C05459=1123.392,111.810,-57.603,-179.804,8.191,149.512
C05460=1123.397,111.561,-57.584,-179.806,8.187,149.511
C05461=1123.401,111.312,-57.565,-179.808,8.184,149.511
C05462=1123.406,111.062,-57.545,-179.809,8.181,149.511
C05463=1123.411,110.813,-57.526,-179.812,8.177,149.510
C05464=1123.416,110.564,-57.506,-179.814,8.173,149.510
C05465=1123.421,110.314,-57.487,-179.817,8.169,149.510
C05466=1123.426,110.066,-57.468,-179.819,8.165,149.510
C05467=1123.430,109.816,-57.448,-179.822,8.161,149.510
C05468=1123.436,109.567,-57.429,-179.824,8.158,149.509
C05469=1123.440,109.318,-57.409,-179.826,8.154,149.509
C05470=1123.444,109.068,-57.390,-179.828,8.150,149.509
C05471=1123.450,108.820,-57.371,-179.830,8.146,149.509
C05472=1123.455,108.570,-57.351,-179.833,8.142,149.508
C05473=1123.460,108.321,-57.332,-179.835,8.138,149.508
C05474=1123.464,108.072,-57.313,-179.838,8.134,149.508
C05475=1123.469,107.823,-57.294,-179.840,8.131,149.508
C05476=1123.474,107.573,-57.274,-179.843,8.126,149.508
C05477=1123.478,107.324,-57.255,-179.845,8.123,149.507
C05478=1123.483,107.075,-57.236,-179.846,8.119,149.507
C05479=1123.488,106.826,-57.216,-179.849,8.115,149.507
C05480=1123.493,106.577,-57.198,-179.851,8.111,149.506
C05481=1123.498,106.327,-57.178,-179.854,8.107,149.506
C05482=1123.503,106.078,-57.159,-179.856,8.103,149.506
C05483=1123.507,105.829,-57.140,-179.857,8.100,149.506
C05484=1123.512,105.580,-57.121,-179.860,8.095,149.505
C05485=1123.516,105.331,-57.102,-179.862,8.092,149.505
C05486=1123.522,105.081,-57.083,-179.864,8.088,149.505
C05487=1123.527,104.832,-57.064,-179.866,8.084,149.505
C05488=1123.531,104.583,-57.045,-179.868,8.080,149.504
C05489=1123.536,104.334,-57.025,-179.870,8.076,149.504
C05490=1123.541,104.084,-57.007,-179.873,8.072,149.504
C05491=1123.546,103.870,-56.991,-179.874,8.069,149.503
C05492=1123.549,103.655,-56.974,-179.876,8.066,149.503
C05493=1123.553,103.441,-56.957,-179.878,8.062,149.503
C05494=1123.557,103.227,-56.941,-179.880,8.058,149.503
C05495=1123.562,103.012,-56.925,-179.881,8.056,149.502
C05496=1123.566,102.798,-56.909,-179.883,8.052,149.502
C05497=1123.570,102.582,-56.892,-179.885,8.048,149.502
C05498=1123.574,102.368,-56.876,-179.886,8.046,149.501
C05499=1123.579,102.119,-56.857,-179.889,8.041,149.501
C05500=1123.583,101.870,-56.838,-179.891,8.037,149.501
C05501=1123.589,101.620,-56.820,-179.892,8.033,149.500
C05502=1123.594,101.372,-56.801,-179.894,8.030,149.500
C05503=1123.598,101.122,-56.781,-179.897,8.025,149.500
C05504=1123.603,100.873,-56.763,-179.899,8.022,149.500
C05505=1123.608,100.623,-56.744,-179.900,8.018,149.499
C05506=1123.613,100.374,-56.726,-179.902,8.014,149.499
C05507=1123.618,100.125,-56.707,-179.905,8.010,149.498
C05508=1123.623,99.875,-56.688,-179.906,8.006,149.498
C05509=1123.627,99.627,-56.669,-179.908,8.002,149.498
C05510=1123.632,99.377,-56.651,-179.910,7.998,149.497
C05511=1123.637,99.128,-56.632,-179.911,7.995,149.497
C05512=1123.642,98.878,-56.613,-179.914,7.990,149.497
C05513=1123.646,98.629,-56.594,-179.916,7.986,149.496
C05514=1123.651,98.380,-56.576,-179.917,7.982,149.496
C05515=1123.657,98.131,-56.557,-179.919,7.979,149.495
C05516=1123.661,97.881,-56.539,-179.921,7.975,149.495
C05517=1123.666,97.632,-56.521,-179.923,7.971,149.495
C05518=1123.671,97.383,-56.501,-179.925,7.967,149.494
C05519=1123.676,97.133,-56.483,-179.926,7.963,149.494
C05520=1123.680,96.885,-56.464,-179.928,7.959,149.494
C05521=1123.686,96.635,-56.446,-179.930,7.955,149.493
C05522=1123.690,96.385,-56.427,-179.932,7.951,149.493
C05523=1123.695,96.137,-56.409,-179.933,7.947,149.492
C05524=1123.700,95.888,-56.391,-179.935,7.944,149.492
C05525=1123.705,95.638,-56.372,-179.936,7.940,149.492
C05526=1123.709,95.389,-56.353,-179.938,7.936,149.491
C05527=1123.714,95.140,-56.335,-179.940,7.932,149.491
C05528=1123.720,94.890,-56.317,-179.942,7.927,149.490
C05529=1123.724,94.640,-56.298,-179.943,7.923,149.490
C05530=1123.729,94.392,-56.279,-179.945,7.919,149.489
C05531=1123.734,94.143,-56.261,-179.947,7.916,149.489
C05532=1123.739,93.894,-56.244,-179.948,7.912,149.489
C05533=1123.744,93.643,-56.225,-179.950,7.908,149.488
C05534=1123.748,93.395,-56.206,-179.951,7.904,149.488
C05535=1123.753,93.146,-56.188,-179.953,7.900,149.487
C05536=1123.758,92.896,-56.170,-179.955,7.896,149.487
C05537=1123.762,92.647,-56.152,-179.956,7.892,149.486
C05538=1123.768,92.397,-56.133,-179.958,7.888,149.486
C05539=1123.773,92.148,-56.115,-179.959,7.884,149.486
C05540=1123.778,91.899,-56.096,-179.961,7.881,149.485
C05541=1123.783,91.650,-56.078,-179.963,7.877,149.485
C05542=1123.787,91.400,-56.060,-179.964,7.873,149.484
C05543=1123.792,91.151,-56.042,-179.966,7.869,149.484
C05544=1123.797,90.902,-56.023,-179.967,7.865,149.483
C05545=1123.802,90.652,-56.005,-179.968,7.862,149.483
C05546=1123.807,90.403,-55.987,-179.970,7.858,149.482
C05547=1123.811,90.189,-55.972,-179.972,7.854,149.482
C05548=1123.815,89.974,-55.956,-179.973,7.851,149.482
C05549=1123.819,89.760,-55.941,-179.974,7.848,149.481
C05550=1123.823,89.545,-55.925,-179.975,7.844,149.481
C05551=1123.828,89.330,-55.909,-179.976,7.841,149.480
C05552=1123.832,89.115,-55.894,-179.978,7.837,149.480
C05553=1123.837,88.901,-55.878,-179.979,7.834,149.480
C05554=1123.840,88.686,-55.862,-179.980,7.831,149.479
C05555=1123.845,88.437,-55.844,-179.981,7.827,149.479
C05556=1123.850,88.187,-55.826,-179.983,7.823,149.478
C05557=1123.854,87.938,-55.808,-179.984,7.819,149.478
C05558=1123.860,87.688,-55.791,-179.986,7.815,149.477
C05559=1123.865,87.439,-55.773,-179.987,7.812,149.477
C05560=1123.870,87.190,-55.755,-179.988,7.808,149.476
C05561=1123.874,86.941,-55.737,-179.990,7.804,149.476
C05562=1123.879,86.692,-55.719,-179.991,7.800,149.475
C05563=1123.884,86.443,-55.701,-179.992,7.796,149.475
C05564=1123.889,86.193,-55.683,-179.993,7.793,149.474
C05565=1123.893,85.943,-55.665,-179.995,7.788,149.474
C05566=1123.898,85.694,-55.647,-179.996,7.784,149.473
C05567=1123.903,85.445,-55.629,-179.998,7.781,149.473
C05568=1123.909,85.195,-55.611,-179.998,7.777,149.472
C05569=1123.913,84.946,-55.593,-180.000,7.773,149.472
C05570=1123.918,84.697,-55.575,179.999,7.769,149.471
C05571=1123.923,84.448,-55.557,179.997,7.765,149.471
C05572=1123.928,84.199,-55.539,179.996,7.762,149.470
C05573=1123.933,83.949,-55.521,179.995,7.758,149.470
C05574=1123.938,83.700,-55.504,179.994,7.754,149.469
C05575=1123.943,83.450,-55.486,179.993,7.751,149.469
C05576=1123.948,83.201,-55.468,179.992,7.746,149.468
C05577=1123.952,82.952,-55.451,179.990,7.742,149.468
C05578=1123.958,82.703,-55.434,179.990,7.739,149.467
C05579=1123.962,82.453,-55.416,179.988,7.735,149.467
C05580=1123.967,82.204,-55.398,179.986,7.731,149.466
C05581=1123.972,81.955,-55.380,179.986,7.728,149.466
C05582=1123.977,81.705,-55.362,179.984,7.724,149.465
C05583=1123.982,81.455,-55.344,179.984,7.720,149.465
C05584=1123.986,81.207,-55.327,179.982,7.716,149.464
C05585=1123.991,80.957,-55.309,179.981,7.712,149.463
C05586=1123.996,80.708,-55.291,179.980,7.709,149.463
C05587=1124.001,80.458,-55.273,179.979,7.705,149.462
C05588=1124.006,80.209,-55.256,179.978,7.702,149.462
C05589=1124.011,79.959,-55.238,179.977,7.697,149.461
C05590=1124.016,79.711,-55.221,179.976,7.694,149.461
C05591=1124.021,79.462,-55.204,179.975,7.690,149.460
C05592=1124.026,79.212,-55.186,179.974,7.687,149.460
C05593=1124.031,78.963,-55.168,179.973,7.682,149.459
C05594=1124.036,78.713,-55.151,179.972,7.679,149.459
C05595=1124.040,78.464,-55.133,179.971,7.675,149.458
C05596=1124.046,78.215,-55.116,179.970,7.672,149.457
C05597=1124.050,77.966,-55.098,179.969,7.668,149.457
C05598=1124.056,77.716,-55.081,179.968,7.664,149.456
C05599=1124.061,77.467,-55.063,179.966,7.660,149.456
C05600=1124.065,77.218,-55.045,179.966,7.657,149.455
C05601=1124.070,76.968,-55.028,179.964,7.653,149.455
C05602=1124.075,76.719,-55.010,179.964,7.649,149.454
C05603=1124.079,76.503,-54.996,179.963,7.646,149.454
C05604=1124.083,76.289,-54.981,179.961,7.642,149.453
C05605=1124.087,76.075,-54.966,179.960,7.639,149.453
C05606=1124.092,75.860,-54.951,179.959,7.635,149.453
C05607=1124.096,75.645,-54.936,179.958,7.632,149.452
C05608=1124.100,75.430,-54.920,179.957,7.629,149.452
C05609=1124.105,75.215,-54.906,179.955,7.625,149.451
C05610=1124.109,75.001,-54.891,179.954,7.622,149.451
C05611=1124.114,74.751,-54.874,179.953,7.618,149.450
C05612=1124.119,74.502,-54.856,179.951,7.614,149.450
C05613=1124.123,74.253,-54.839,179.950,7.610,149.450
C05614=1124.128,74.003,-54.821,179.948,7.606,149.449
C05615=1124.133,73.754,-54.804,179.947,7.602,149.448
C05616=1124.138,73.504,-54.787,179.945,7.598,149.448
C05617=1124.143,73.255,-54.769,179.944,7.594,149.448
C05618=1124.149,73.006,-54.752,179.942,7.590,149.447
C05619=1124.153,72.756,-54.736,179.941,7.586,149.447
C05620=1124.158,72.507,-54.718,179.939,7.582,149.446
C05621=1124.162,72.258,-54.701,179.938,7.578,149.446
C05622=1124.168,72.008,-54.684,179.937,7.574,149.445
C05623=1124.173,71.759,-54.666,179.935,7.570,149.445
C05624=1124.177,71.509,-54.649,179.934,7.566,149.444
C05625=1124.183,71.260,-54.632,179.932,7.562,149.444
C05626=1124.187,71.011,-54.615,179.931,7.558,149.443
C05627=1124.192,70.762,-54.598,179.929,7.554,149.443
C05628=1124.197,70.512,-54.581,179.928,7.550,149.442
C05629=1124.202,70.262,-54.564,179.926,7.546,149.442
C05630=1124.207,70.014,-54.546,179.926,7.543,149.441
C05631=1124.212,69.764,-54.529,179.924,7.539,149.441
C05632=1124.217,69.514,-54.512,179.923,7.535,149.440
C05633=1124.222,69.265,-54.496,179.921,7.531,149.440
C05634=1124.227,69.015,-54.478,179.920,7.527,149.439
C05635=1124.232,68.767,-54.461,179.918,7.523,149.439
C05636=1124.237,68.517,-54.444,179.917,7.519,149.438
C05637=1124.241,68.268,-54.427,179.916,7.515,149.438
C05638=1124.247,68.018,-54.410,179.914,7.511,149.437
C05639=1124.252,67.769,-54.394,179.912,7.507,149.437
C05640=1124.256,67.520,-54.377,179.911,7.503,149.436
C05641=1124.261,67.270,-54.360,179.910,7.499,149.436
C05642=1124.265,67.021,-54.342,179.908,7.495,149.435
C05643=1124.271,66.772,-54.326,179.907,7.491,149.435
C05644=1124.276,66.522,-54.309,179.906,7.487,149.434
C05645=1124.281,66.273,-54.292,179.904,7.483,149.434
C05646=1124.285,66.023,-54.275,179.903,7.478,149.433
C05647=1124.291,65.774,-54.259,179.901,7.475,149.433
C05648=1124.296,65.525,-54.241,179.900,7.471,149.432
C05649=1124.300,65.275,-54.225,179.899,7.466,149.432
C05650=1124.306,65.026,-54.208,179.898,7.463,149.431
C05651=1124.311,64.777,-54.191,179.896,7.459,149.431
C05652=1124.315,64.527,-54.174,179.895,7.455,149.430
C05653=1124.321,64.278,-54.158,179.893,7.451,149.430
C05654=1124.325,64.028,-54.141,179.892,7.447,149.429
C05655=1124.330,63.779,-54.124,179.891,7.443,149.429
C05656=1124.335,63.529,-54.107,179.889,7.439,149.428
C05657=1124.340,63.280,-54.091,179.888,7.435,149.428
C05658=1124.345,63.031,-54.074,179.887,7.431,149.427
C05659=1124.350,62.816,-54.060,179.886,7.428,149.427
C05660=1124.353,62.601,-54.046,179.884,7.424,149.426
C05661=1124.358,62.386,-54.031,179.883,7.421,149.426
C05662=1124.362,62.172,-54.017,179.882,7.417,149.426
C05663=1124.366,61.956,-54.003,179.881,7.414,149.425
C05664=1124.370,61.741,-53.988,179.880,7.411,149.425
C05665=1124.375,61.527,-53.973,179.878,7.407,149.424
C05666=1124.379,61.312,-53.959,179.877,7.403,149.424
C05667=1124.385,61.062,-53.943,179.876,7.400,149.423
C05668=1124.389,60.813,-53.927,179.874,7.395,149.423
C05669=1124.394,60.563,-53.910,179.873,7.391,149.422
C05670=1124.399,60.315,-53.894,179.871,7.387,149.422
C05671=1124.404,60.065,-53.876,179.870,7.383,149.421
C05672=1124.409,59.816,-53.860,179.869,7.379,149.421
C05673=1124.414,59.566,-53.844,179.868,7.375,149.420
C05674=1124.418,59.317,-53.827,179.866,7.371,149.420
C05675=1124.423,59.068,-53.811,179.864,7.367,149.419
C05676=1124.429,58.818,-53.794,179.863,7.363,149.419
C05677=1124.434,58.569,-53.778,179.862,7.359,149.418
C05678=1124.438,58.319,-53.762,179.861,7.355,149.418
C05679=1124.444,58.070,-53.745,179.859,7.351,149.417
C05680=1124.448,57.820,-53.729,179.858,7.348,149.417
C05681=1124.453,57.571,-53.713,179.857,7.343,149.416
C05682=1124.459,57.322,-53.696,179.856,7.339,149.416
C05683=1124.463,57.071,-53.680,179.854,7.335,149.415
C05684=1124.469,56.823,-53.663,179.853,7.331,149.415
C05685=1124.473,56.573,-53.647,179.852,7.327,149.414
C05686=1124.478,56.324,-53.631,179.850,7.323,149.414
C05687=1124.483,56.074,-53.615,179.849,7.319,149.413
C05688=1124.488,55.826,-53.598,179.848,7.315,149.412
C05689=1124.493,55.575,-53.582,179.846,7.311,149.412
C05690=1124.499,55.326,-53.565,179.845,7.307,149.411
C05691=1124.503,55.076,-53.549,179.843,7.303,149.411
C05692=1124.508,54.827,-53.533,179.842,7.298,149.410
C05693=1124.513,54.577,-53.517,179.841,7.294,149.410
C05694=1124.518,54.329,-53.501,179.840,7.290,149.409
C05695=1124.523,54.079,-53.484,179.838,7.286,149.409
C05696=1124.528,53.830,-53.469,179.837,7.282,149.408
C05697=1124.533,53.580,-53.452,179.835,7.278,149.408
C05698=1124.538,53.331,-53.436,179.834,7.274,149.407
C05699=1124.542,53.081,-53.420,179.833,7.271,149.407
C05700=1124.548,52.832,-53.404,179.832,7.266,149.406
C05701=1124.552,52.582,-53.387,179.831,7.262,149.406
C05702=1124.558,52.333,-53.372,179.830,7.258,149.405
C05703=1124.563,52.084,-53.356,179.828,7.254,149.405
C05704=1124.568,51.834,-53.340,179.827,7.250,149.404
C05705=1124.573,51.585,-53.324,179.825,7.246,149.403
C05706=1124.577,51.335,-53.307,179.824,7.242,149.403
C05707=1124.583,51.086,-53.292,179.823,7.238,149.402
C05708=1124.587,50.836,-53.275,179.822,7.233,149.402
C05709=1124.593,50.587,-53.259,179.820,7.230,149.401
C05710=1124.598,50.338,-53.244,179.819,7.225,149.401
C05711=1124.603,50.088,-53.227,179.817,7.221,149.400
C05712=1124.608,49.839,-53.212,179.816,7.217,149.400
C05713=1124.613,49.589,-53.196,179.815,7.213,149.399
C05714=1124.618,49.340,-53.179,179.814,7.209,149.398
C05715=1124.622,49.125,-53.166,179.813,7.206,149.398
C05716=1124.626,48.910,-53.152,179.811,7.202,149.398
C05717=1124.630,48.695,-53.139,179.811,7.198,149.397
C05718=1124.634,48.480,-53.125,179.810,7.195,149.397
C05719=1124.639,48.265,-53.111,179.808,7.191,149.396
C05720=1124.643,48.050,-53.098,179.807,7.188,149.396
C05721=1124.648,47.835,-53.084,179.806,7.184,149.395
C05722=1124.652,47.620,-53.071,179.805,7.181,149.395
C05723=1124.657,47.371,-53.054,179.804,7.177,149.394
C05724=1124.662,47.121,-53.039,179.803,7.172,149.394
C05725=1124.667,46.872,-53.024,179.802,7.168,149.393
C05726=1124.672,46.622,-53.008,179.800,7.164,149.392
C05727=1124.677,46.373,-52.991,179.799,7.160,149.392
C05728=1124.682,46.124,-52.976,179.798,7.156,149.391
C05729=1124.687,45.874,-52.960,179.796,7.152,149.391
C05730=1124.692,45.624,-52.944,179.795,7.147,149.390
C05731=1124.697,45.375,-52.929,179.794,7.143,149.390
C05732=1124.702,45.125,-52.913,179.793,7.139,149.389
C05733=1124.707,44.876,-52.897,179.792,7.135,149.388
C05734=1124.712,44.627,-52.881,179.790,7.131,149.388
C05735=1124.716,44.377,-52.866,179.789,7.127,149.387
C05736=1124.722,44.128,-52.850,179.788,7.122,149.387
C05737=1124.727,43.878,-52.835,179.786,7.118,149.386
C05738=1124.732,43.629,-52.819,179.785,7.114,149.386
C05739=1124.736,43.379,-52.804,179.784,7.110,149.385
C05740=1124.742,43.130,-52.788,179.783,7.106,149.385
C05741=1124.747,42.880,-52.773,179.782,7.102,149.384
C05742=1124.753,42.631,-52.757,179.781,7.098,149.383
C05743=1124.757,42.381,-52.742,179.780,7.094,149.383
C05744=1124.762,42.132,-52.726,179.779,7.090,149.382
C05745=1124.767,41.882,-52.711,179.777,7.085,149.382
C05746=1124.772,41.633,-52.696,179.776,7.082,149.381
C05747=1124.777,41.383,-52.680,179.775,7.077,149.380
C05748=1124.782,41.134,-52.664,179.774,7.073,149.380
C05749=1124.787,40.885,-52.649,179.773,7.069,149.379
C05750=1124.792,40.635,-52.634,179.771,7.065,149.379
C05751=1124.797,40.385,-52.618,179.770,7.060,149.378
C05752=1124.802,40.136,-52.603,179.769,7.056,149.377
C05753=1124.807,39.887,-52.587,179.768,7.052,149.377
C05754=1124.813,39.637,-52.571,179.766,7.048,149.376
C05755=1124.817,39.388,-52.556,179.765,7.044,149.376
C05756=1124.823,39.139,-52.541,179.764,7.039,149.375
C05757=1124.827,38.889,-52.525,179.763,7.035,149.374
C05758=1124.832,38.640,-52.510,179.762,7.031,149.374
C05759=1124.837,38.390,-52.494,179.761,7.027,149.373
C05760=1124.842,38.141,-52.480,179.759,7.022,149.373
C05761=1124.848,37.891,-52.464,179.758,7.018,149.372
C05762=1124.852,37.642,-52.449,179.757,7.014,149.371
C05763=1124.857,37.392,-52.433,179.756,7.010,149.371
C05764=1124.863,37.143,-52.418,179.755,7.006,149.370
C05765=1124.868,36.893,-52.404,179.754,7.001,149.370
C05766=1124.873,36.643,-52.388,179.753,6.997,149.369
C05767=1124.878,36.394,-52.373,179.752,6.993,149.368
C05768=1124.883,36.145,-52.357,179.750,6.988,149.368
C05769=1124.888,35.896,-52.342,179.749,6.984,149.367
C05770=1124.893,35.645,-52.327,179.748,6.980,149.367
C05771=1124.897,35.430,-52.314,179.747,6.976,149.366
C05772=1124.902,35.215,-52.301,179.746,6.973,149.366
C05773=1124.905,35.001,-52.288,179.745,6.969,149.365
C05774=1124.910,34.786,-52.275,179.744,6.965,149.364
C05775=1124.914,34.571,-52.262,179.743,6.962,149.364
C05776=1124.919,34.356,-52.249,179.742,6.958,149.363
C05777=1124.923,34.141,-52.236,179.741,6.954,149.363
C05778=1124.928,33.926,-52.223,179.740,6.950,149.362
C05779=1124.933,33.676,-52.209,179.739,6.946,149.362
C05780=1124.938,33.427,-52.193,179.738,6.942,149.361
C05781=1124.943,33.178,-52.178,179.737,6.937,149.360
C05782=1124.947,32.927,-52.163,179.736,6.933,149.360
C05783=1124.953,32.678,-52.148,179.735,6.929,149.359
C05784=1124.957,32.429,-52.133,179.733,6.925,149.359
C05785=1124.963,32.179,-52.118,179.732,6.920,149.358
C05786=1124.968,31.930,-52.103,179.731,6.916,149.357
C05787=1124.973,31.680,-52.089,179.730,6.912,149.357
C05788=1124.978,31.430,-52.073,179.729,6.908,149.356
C05789=1124.983,31.181,-52.059,179.728,6.903,149.355
C05790=1124.988,30.931,-52.043,179.727,6.899,149.355
C05791=1124.993,30.682,-52.028,179.726,6.895,149.354
C05792=1124.998,30.433,-52.014,179.725,6.890,149.353
C05793=1125.003,30.183,-51.998,179.724,6.886,149.353
C05794=1125.008,29.933,-51.984,179.722,6.882,149.352
C05795=1125.013,29.684,-51.969,179.721,6.877,149.352
C05796=1125.019,29.434,-51.954,179.720,6.873,149.351
C05797=1125.023,29.185,-51.939,179.719,6.869,149.350
C05798=1125.028,28.935,-51.925,179.718,6.864,149.350
C05799=1125.034,28.686,-51.909,179.717,6.860,149.349
C05800=1125.038,28.436,-51.895,179.716,6.856,149.348
C05801=1125.043,28.187,-51.881,179.715,6.851,149.348
C05802=1125.048,27.938,-51.866,179.714,6.847,149.347
C05803=1125.054,27.688,-51.851,179.713,6.843,149.346
C05804=1125.058,27.438,-51.836,179.712,6.839,149.346
C05805=1125.063,27.189,-51.822,179.711,6.834,149.345
C05806=1125.069,26.939,-51.807,179.710,6.829,149.344
C05807=1125.074,26.690,-51.792,179.709,6.824,149.344
C05808=1125.079,26.440,-51.777,179.708,6.820,149.343
C05809=1125.084,26.191,-51.764,179.707,6.816,149.342
C05810=1125.089,25.942,-51.749,179.705,6.811,149.342
C05811=1125.095,25.692,-51.734,179.704,6.807,149.341
C05812=1125.100,25.442,-51.719,179.703,6.803,149.340
C05813=1125.104,25.193,-51.704,179.702,6.798,149.340
C05814=1125.109,24.943,-51.690,179.701,6.794,149.339
C05815=1125.115,24.693,-51.675,179.701,6.789,149.338
C05816=1125.119,24.444,-51.660,179.700,6.785,149.337
C05817=1125.124,24.194,-51.646,179.699,6.781,149.337
C05818=1125.129,23.945,-51.632,179.698,6.777,149.336
C05819=1125.134,23.695,-51.617,179.696,6.772,149.335
C05820=1125.140,23.447,-51.603,179.695,6.768,149.335
C05821=1125.145,23.197,-51.588,179.695,6.763,149.334
C05822=1125.150,22.947,-51.574,179.694,6.759,149.333
C05823=1125.155,22.697,-51.559,179.692,6.754,149.333
C05824=1125.160,22.447,-51.545,179.691,6.749,149.332
C05825=1125.165,22.198,-51.530,179.690,6.745,149.331
C05826=1125.170,21.949,-51.516,179.689,6.740,149.331
C05827=1125.175,21.733,-51.504,179.689,6.737,149.330
C05828=1125.179,21.518,-51.491,179.688,6.733,149.329
C05829=1125.183,21.303,-51.479,179.687,6.729,149.329
C05830=1125.187,21.088,-51.466,179.686,6.725,149.328
C05831=1125.192,20.873,-51.454,179.686,6.722,149.327
C05832=1125.196,20.658,-51.442,179.684,6.718,149.327
C05833=1125.201,20.442,-51.429,179.684,6.714,149.326
C05834=1125.205,20.228,-51.417,179.683,6.710,149.326
C05835=1125.210,19.978,-51.403,179.682,6.705,149.325
C05836=1125.215,19.729,-51.389,179.681,6.701,149.324
C05837=1125.220,19.479,-51.375,179.680,6.696,149.324
C05838=1125.225,19.230,-51.360,179.679,6.692,149.323
C05839=1125.230,18.980,-51.346,179.678,6.688,149.322
C05840=1125.235,18.730,-51.332,179.677,6.683,149.321
C05841=1125.241,18.481,-51.318,179.676,6.678,149.321
C05842=1125.246,18.232,-51.304,179.675,6.674,149.320
C05843=1125.251,17.982,-51.289,179.674,6.669,149.319
C05844=1125.256,17.732,-51.275,179.673,6.665,149.319
C05845=1125.261,17.483,-51.261,179.672,6.660,149.318
C05846=1125.266,17.233,-51.247,179.671,6.656,149.317
C05847=1125.271,16.984,-51.233,179.670,6.651,149.316
C05848=1125.276,16.734,-51.218,179.670,6.647,149.315
C05849=1125.282,16.485,-51.204,179.669,6.642,149.315
C05850=1125.287,16.235,-51.190,179.667,6.637,149.314
C05851=1125.291,15.986,-51.176,179.667,6.632,149.313
C05852=1125.296,15.736,-51.162,179.666,6.628,149.313
C05853=1125.302,15.487,-51.148,179.665,6.623,149.312
C05854=1125.307,15.237,-51.133,179.664,6.619,149.311
C05855=1125.312,14.987,-51.119,179.663,6.615,149.310
C05856=1125.317,14.738,-51.105,179.662,6.610,149.310
C05857=1125.323,14.488,-51.092,179.661,6.606,149.309
C05858=1125.327,14.239,-51.078,179.660,6.600,149.308
C05859=1125.332,13.989,-51.064,179.659,6.596,149.307
C05860=1125.337,13.740,-51.050,179.659,6.591,149.307
C05861=1125.342,13.490,-51.035,179.658,6.587,149.306
C05862=1125.347,13.241,-51.021,179.657,6.582,149.305
C05863=1125.353,12.991,-51.008,179.656,6.578,149.304
C05864=1125.358,12.741,-50.994,179.655,6.573,149.304
C05865=1125.362,12.492,-50.980,179.654,6.568,149.303
C05866=1125.368,12.243,-50.966,179.653,6.563,149.302
C05867=1125.373,11.992,-50.953,179.652,6.559,149.301
C05868=1125.378,11.743,-50.938,179.652,6.554,149.300
C05869=1125.384,11.494,-50.924,179.651,6.549,149.300
C05870=1125.389,11.244,-50.910,179.650,6.545,149.299
C05871=1125.393,10.994,-50.897,179.649,6.540,149.298
C05872=1125.399,10.745,-50.883,179.648,6.535,149.297
C05873=1125.404,10.495,-50.869,179.647,6.531,149.297
C05874=1125.410,10.246,-50.856,179.646,6.526,149.296
C05875=1125.414,9.996,-50.842,179.646,6.522,149.295
C05876=1125.419,9.747,-50.828,179.645,6.517,149.294
C05877=1125.425,9.497,-50.815,179.644,6.512,149.293
C05878=1125.430,9.247,-50.800,179.643,6.507,149.293
C05879=1125.434,8.999,-50.787,179.642,6.502,149.292
C05880=1125.440,8.748,-50.773,179.641,6.498,149.291
C05881=1125.445,8.498,-50.759,179.641,6.493,149.290
C05882=1125.450,8.249,-50.746,179.640,6.488,149.289
C05883=1125.455,8.034,-50.734,179.639,6.484,149.289
C05884=1125.459,7.818,-50.723,179.639,6.481,149.288
C05885=1125.463,7.603,-50.711,179.639,6.477,149.287
C05886=1125.467,7.388,-50.699,179.638,6.472,149.286
C05887=1125.473,7.173,-50.687,179.638,6.468,149.286
C05888=1125.477,6.958,-50.676,179.638,6.465,149.285
C05889=1125.481,6.742,-50.664,179.637,6.461,149.284
C05890=1125.485,6.527,-50.652,179.637,6.457,149.283
C05891=1125.491,6.278,-50.638,179.637,6.453,149.282
C05892=1125.495,6.028,-50.625,179.636,6.448,149.282
C05893=1125.500,5.778,-50.611,179.635,6.444,149.281
C05894=1125.506,5.529,-50.598,179.635,6.439,149.280
C05895=1125.510,5.279,-50.584,179.635,6.435,149.279
C05896=1125.516,5.030,-50.571,179.634,6.430,149.278
C05897=1125.521,4.780,-50.557,179.634,6.426,149.277
C05898=1125.526,4.531,-50.544,179.633,6.421,149.277
C05899=1125.531,4.281,-50.530,179.633,6.416,149.276
C05900=1125.536,4.032,-50.517,179.632,6.413,149.275
C05901=1125.541,3.782,-50.503,179.632,6.408,149.274
C05902=1125.547,3.532,-50.490,179.631,6.403,149.273
C05903=1125.551,3.283,-50.476,179.631,6.398,149.272
C05904=1125.557,3.033,-50.463,179.630,6.394,149.271
C05905=1125.562,2.783,-50.450,179.630,6.390,149.271
C05906=1125.567,2.534,-50.436,179.629,6.385,149.270
C05907=1125.572,2.284,-50.423,179.629,6.381,149.269
C05908=1125.577,2.035,-50.409,179.628,6.376,149.268
C05909=1125.583,1.785,-50.396,179.627,6.371,149.267
C05910=1125.588,1.536,-50.383,179.628,6.367,149.266
C05911=1125.593,1.287,-50.369,179.627,6.363,149.266
C05912=1125.598,1.037,-50.356,179.626,6.358,149.265
C05913=1125.604,0.787,-50.343,179.626,6.354,149.264
C05914=1125.608,0.538,-50.329,179.625,6.349,149.263
C05915=1125.614,0.288,-50.316,179.624,6.345,149.262
C05916=1125.618,0.038,-50.303,179.624,6.341,149.262
C05917=1125.624,-0.212,-50.290,179.624,6.336,149.261
C05918=1125.628,-0.461,-50.276,179.623,6.331,149.260
C05919=1125.634,-0.711,-50.263,179.622,6.327,149.259
C05920=1125.639,-0.960,-50.250,179.621,6.322,149.258
C05921=1125.644,-1.210,-50.236,179.621,6.317,149.257
C05922=1125.649,-1.459,-50.224,179.621,6.313,149.256
C05923=1125.654,-1.709,-50.211,179.620,6.309,149.256
C05924=1125.660,-1.959,-50.197,179.619,6.304,149.255
C05925=1125.665,-2.208,-50.185,179.619,6.300,149.254
C05926=1125.670,-2.458,-50.171,179.618,6.295,149.253
C05927=1125.675,-2.707,-50.158,179.617,6.291,149.253
C05928=1125.680,-2.957,-50.144,179.617,6.286,149.252
C05929=1125.685,-3.207,-50.132,179.616,6.281,149.251
C05930=1125.691,-3.456,-50.119,179.616,6.278,149.250
C05931=1125.695,-3.706,-50.105,179.615,6.273,149.249
C05932=1125.701,-3.955,-50.092,179.615,6.268,149.248
C05933=1125.706,-4.205,-50.079,179.614,6.264,149.248
C05934=1125.711,-4.455,-50.066,179.613,6.259,149.247
C05935=1125.716,-4.704,-50.054,179.613,6.254,149.246
C05936=1125.722,-4.954,-50.040,179.612,6.250,149.245
C05937=1125.726,-5.204,-50.027,179.611,6.245,149.244
C05938=1125.732,-5.453,-50.014,179.611,6.241,149.243
C05939=1125.736,-5.668,-50.003,179.611,6.237,149.243
C05940=1125.740,-5.884,-49.992,179.610,6.233,149.242
C05941=1125.745,-6.099,-49.981,179.609,6.229,149.241
C05942=1125.749,-6.314,-49.969,179.609,6.225,149.241
C05943=1125.754,-6.530,-49.958,179.608,6.221,149.240
C05944=1125.758,-6.744,-49.947,179.608,6.217,149.239
C05945=1125.763,-6.960,-49.936,179.607,6.214,149.239
C05946=1125.767,-7.176,-49.924,179.606,6.209,149.238
C05947=1125.772,-7.425,-49.912,179.606,6.205,149.237
C05948=1125.777,-7.674,-49.899,179.605,6.200,149.236
C05949=1125.783,-7.924,-49.886,179.604,6.196,149.236
C05950=1125.788,-8.174,-49.873,179.604,6.191,149.235
C05951=1125.793,-8.423,-49.860,179.603,6.187,149.234
C05952=1125.799,-8.673,-49.847,179.602,6.182,149.233
C05953=1125.803,-8.923,-49.834,179.602,6.177,149.232
C05954=1125.809,-9.173,-49.822,179.601,6.173,149.232
C05955=1125.814,-9.422,-49.810,179.600,6.168,149.231
C05956=1125.820,-9.672,-49.796,179.600,6.163,149.230
C05957=1125.824,-9.922,-49.783,179.599,6.159,149.229
C05958=1125.829,-10.171,-49.771,179.598,6.154,149.228
C05959=1125.834,-10.420,-49.758,179.598,6.149,149.227
C05960=1125.840,-10.670,-49.746,179.597,6.145,149.227
C05961=1125.845,-10.920,-49.732,179.596,6.140,149.226
C05962=1125.850,-11.169,-49.719,179.596,6.136,149.225
C05963=1125.855,-11.419,-49.707,179.595,6.131,149.224
C05964=1125.860,-11.669,-49.695,179.594,6.127,149.223
C05965=1125.865,-11.919,-49.682,179.594,6.122,149.222
C05966=1125.870,-12.168,-49.669,179.593,6.118,149.222
C05967=1125.876,-12.418,-49.656,179.592,6.113,149.221
C05968=1125.881,-12.667,-49.644,179.592,6.108,149.220
C05969=1125.886,-12.916,-49.631,179.591,6.104,149.219
C05970=1125.891,-13.167,-49.619,179.590,6.099,149.218
C05971=1125.896,-13.416,-49.606,179.590,6.094,149.218
C05972=1125.901,-13.665,-49.594,179.589,6.090,149.217
C05973=1125.906,-13.915,-49.581,179.588,6.085,149.216
C05974=1125.913,-14.165,-49.568,179.588,6.080,149.215
C05975=1125.917,-14.415,-49.555,179.587,6.076,149.214
C05976=1125.922,-14.664,-49.543,179.587,6.071,149.214
C05977=1125.927,-14.914,-49.530,179.586,6.067,149.213
C05978=1125.933,-15.164,-49.518,179.584,6.062,149.212
C05979=1125.938,-15.413,-49.506,179.584,6.057,149.211
C05980=1125.943,-15.662,-49.493,179.583,6.052,149.210
C05981=1125.948,-15.913,-49.481,179.582,6.048,149.210
C05982=1125.953,-16.162,-49.468,179.582,6.043,149.209
C05983=1125.958,-16.412,-49.456,179.581,6.038,149.208
C05984=1125.964,-16.661,-49.444,179.580,6.034,149.207
C05985=1125.969,-16.911,-49.431,179.580,6.029,149.206
C05986=1125.974,-17.160,-49.419,179.579,6.024,149.205
C05987=1125.979,-17.410,-49.407,179.578,6.019,149.205
C05988=1125.984,-17.659,-49.394,179.577,6.015,149.204
C05989=1125.989,-17.909,-49.382,179.577,6.010,149.203
C05990=1125.994,-18.159,-49.369,179.576,6.005,149.202
C05991=1125.999,-18.409,-49.357,179.575,6.001,149.201
C05992=1126.005,-18.659,-49.345,179.574,5.995,149.201
C05993=1126.010,-18.908,-49.332,179.574,5.990,149.200
C05994=1126.015,-19.158,-49.320,179.573,5.986,149.199
C05995=1126.020,-19.373,-49.310,179.572,5.981,149.198
C05996=1126.025,-19.589,-49.299,179.572,5.978,149.197
C05997=1126.029,-19.804,-49.289,179.571,5.973,149.197
C05998=1126.033,-20.019,-49.277,179.570,5.969,149.196
C05999=1126.038,-20.234,-49.267,179.570,5.965,149.195
C06000=1126.042,-20.450,-49.256,179.569,5.961,149.195
C06001=1126.047,-20.665,-49.246,179.569,5.957,149.194
C06002=1126.051,-20.881,-49.235,179.568,5.953,149.193
C06003=1126.057,-21.131,-49.223,179.567,5.948,149.192
C06004=1126.062,-21.380,-49.211,179.566,5.943,149.191
C06005=1126.067,-21.630,-49.199,179.565,5.938,149.191
C06006=1126.073,-21.880,-49.187,179.565,5.934,149.190
C06007=1126.078,-22.129,-49.174,179.564,5.929,149.189
C06008=1126.083,-22.379,-49.162,179.563,5.923,149.188
C06009=1126.088,-22.628,-49.150,179.563,5.919,149.187
C06010=1126.093,-22.878,-49.139,179.562,5.914,149.187
C06011=1126.098,-23.128,-49.127,179.561,5.909,149.186
C06012=1126.103,-23.377,-49.114,179.560,5.904,149.185
C06013=1126.109,-23.627,-49.102,179.560,5.899,149.184
C06014=1126.114,-23.877,-49.090,179.559,5.894,149.183
C06015=1126.119,-24.126,-49.078,179.558,5.889,149.182
C06016=1126.125,-24.376,-49.066,179.557,5.885,149.181
C06017=1126.130,-24.626,-49.054,179.556,5.879,149.181
C06018=1126.135,-24.875,-49.042,179.556,5.874,149.180
C06019=1126.140,-25.125,-49.030,179.555,5.870,149.179
C06020=1126.146,-25.375,-49.018,179.554,5.864,149.178
C06021=1126.151,-25.624,-49.006,179.553,5.860,149.177
C06022=1126.155,-25.874,-48.994,179.553,5.855,149.176
C06023=1126.161,-26.124,-48.982,179.553,5.850,149.175
C06024=1126.167,-26.373,-48.971,179.554,5.846,149.174
C06025=1126.172,-26.623,-48.958,179.555,5.842,149.173
C06026=1126.177,-26.872,-48.947,179.556,5.838,149.172
C06027=1126.182,-27.122,-48.935,179.557,5.834,149.171
C06028=1126.187,-27.372,-48.923,179.558,5.831,149.169
C06029=1126.193,-27.621,-48.911,179.558,5.826,149.168
C06030=1126.197,-27.871,-48.899,179.560,5.823,149.167
C06031=1126.203,-28.121,-48.887,179.560,5.818,149.166
C06032=1126.208,-28.371,-48.876,179.560,5.814,149.165
C06033=1126.213,-28.620,-48.864,179.562,5.811,149.164
C06034=1126.218,-28.870,-48.852,179.562,5.806,149.163
C06035=1126.223,-29.120,-48.840,179.562,5.803,149.162
C06036=1126.229,-29.370,-48.828,179.563,5.798,149.161
C06037=1126.234,-29.619,-48.817,179.563,5.794,149.160
C06038=1126.240,-29.869,-48.805,179.564,5.790,149.159
C06039=1126.245,-30.118,-48.792,179.564,5.786,149.158
C06040=1126.250,-30.368,-48.781,179.564,5.782,149.157
C06041=1126.255,-30.617,-48.769,179.565,5.778,149.156
C06042=1126.260,-30.867,-48.757,179.565,5.774,149.155
C06043=1126.266,-31.117,-48.745,179.564,5.769,149.154
C06044=1126.270,-31.367,-48.734,179.564,5.765,149.153
C06045=1126.275,-31.616,-48.722,179.565,5.761,149.152
C06046=1126.281,-31.866,-48.710,179.565,5.756,149.151
C06047=1126.286,-32.115,-48.699,179.565,5.752,149.150
C06048=1126.292,-32.365,-48.687,179.565,5.748,149.149
C06049=1126.297,-32.615,-48.675,179.564,5.743,149.148
C06050=1126.302,-32.865,-48.664,179.564,5.739,149.148
C06051=1126.307,-33.080,-48.653,179.564,5.735,149.147
C06052=1126.311,-33.296,-48.643,179.564,5.731,149.146
C06053=1126.315,-33.511,-48.633,179.563,5.728,149.145
C06054=1126.320,-33.727,-48.623,179.563,5.724,149.145
C06055=1126.324,-33.942,-48.613,179.563,5.720,149.144
C06056=1126.329,-34.157,-48.603,179.562,5.716,149.143
C06057=1126.333,-34.374,-48.593,179.562,5.712,149.142
C06058=1126.338,-34.588,-48.583,179.561,5.708,149.142
C06059=1126.343,-34.838,-48.571,179.561,5.703,149.141
C06060=1126.348,-35.088,-48.560,179.560,5.698,149.140
C06061=1126.354,-35.337,-48.548,179.559,5.694,149.139
C06062=1126.359,-35.587,-48.536,179.559,5.689,149.138
C06063=1126.364,-35.837,-48.525,179.558,5.685,149.138
C06064=1126.370,-36.087,-48.513,179.557,5.680,149.137
C06065=1126.374,-36.336,-48.502,179.556,5.676,149.136
C06066=1126.380,-36.586,-48.490,179.555,5.670,149.135
C06067=1126.385,-36.835,-48.479,179.554,5.666,149.135
C06068=1126.390,-37.085,-48.467,179.553,5.660,149.134
C06069=1126.396,-37.335,-48.455,179.552,5.656,149.133
C06070=1126.400,-37.585,-48.444,179.551,5.650,149.132
C06071=1126.407,-37.834,-48.433,179.550,5.646,149.131
C06072=1126.411,-38.084,-48.421,179.549,5.641,149.131
C06073=1126.417,-38.334,-48.410,179.548,5.635,149.130
C06074=1126.422,-38.584,-48.399,179.546,5.630,149.129
C06075=1126.428,-38.833,-48.387,179.545,5.625,149.129
C06076=1126.432,-39.083,-48.376,179.544,5.620,149.128
C06077=1126.438,-39.333,-48.364,179.543,5.615,149.127
C06078=1126.443,-39.581,-48.353,179.541,5.610,149.126
C06079=1126.448,-39.832,-48.343,179.540,5.604,149.125
C06080=1126.453,-40.082,-48.331,179.538,5.598,149.125
C06081=1126.458,-40.331,-48.319,179.537,5.593,149.124
C06082=1126.464,-40.581,-48.308,179.535,5.588,149.123
C06083=1126.469,-40.830,-48.297,179.533,5.582,149.123
C06084=1126.475,-41.081,-48.285,179.532,5.577,149.122
C06085=1126.480,-41.330,-48.274,179.530,5.571,149.121
C06086=1126.485,-41.579,-48.263,179.528,5.565,149.121
C06087=1126.490,-41.830,-48.252,179.527,5.560,149.120
C06088=1126.496,-42.079,-48.241,179.525,5.554,149.119
C06089=1126.500,-42.328,-48.230,179.523,5.548,149.118
C06090=1126.506,-42.579,-48.219,179.521,5.542,149.118
C06091=1126.511,-42.828,-48.208,179.519,5.537,149.117
C06092=1126.516,-43.077,-48.196,179.517,5.531,149.116
C06093=1126.522,-43.327,-48.186,179.516,5.525,149.115
C06094=1126.527,-43.577,-48.174,179.517,5.521,149.114
C06095=1126.532,-43.827,-48.164,179.517,5.516,149.113
C06096=1126.538,-44.076,-48.152,179.517,5.512,149.112
C06097=1126.543,-44.326,-48.141,179.517,5.507,149.111
C06098=1126.548,-44.576,-48.130,179.518,5.502,149.110
C06099=1126.553,-44.825,-48.119,179.518,5.497,149.109
C06100=1126.559,-45.076,-48.108,179.518,5.492,149.108
C06101=1126.564,-45.325,-48.097,179.518,5.488,149.107
C06102=1126.569,-45.575,-48.087,179.518,5.483,149.106
C06103=1126.574,-45.824,-48.076,179.519,5.479,149.104
C06104=1126.580,-46.074,-48.065,179.518,5.474,149.104
C06105=1126.585,-46.324,-48.053,179.518,5.469,149.102
C06106=1126.590,-46.574,-48.043,179.519,5.464,149.101
C06107=1126.595,-46.789,-48.034,179.519,5.461,149.100
C06108=1126.599,-47.005,-48.024,179.519,5.457,149.099
C06109=1126.603,-47.220,-48.014,179.520,5.453,149.099
C06110=1126.608,-47.436,-48.005,179.520,5.449,149.098
C06111=1126.613,-47.651,-47.996,179.519,5.444,149.097
C06112=1126.617,-47.867,-47.986,179.520,5.440,149.096
C06113=1126.622,-48.082,-47.977,179.520,5.436,149.095
C06114=1126.627,-48.298,-47.968,179.520,5.432,149.094
C06115=1126.632,-48.548,-47.957,179.521,5.428,149.093
C06116=1126.638,-48.797,-47.946,179.521,5.423,149.092
C06117=1126.643,-49.047,-47.935,179.521,5.417,149.091
C06118=1126.647,-49.297,-47.924,179.521,5.413,149.090
C06119=1126.653,-49.547,-47.914,179.521,5.408,149.089
C06120=1126.658,-49.797,-47.903,179.522,5.404,149.087
C06121=1126.664,-50.046,-47.892,179.522,5.399,149.086
C06122=1126.669,-50.296,-47.881,179.522,5.395,149.085
C06123=1126.674,-50.545,-47.870,179.522,5.390,149.084
C06124=1126.679,-50.795,-47.859,179.522,5.385,149.083
C06125=1126.685,-51.045,-47.849,179.522,5.381,149.082
C06126=1126.690,-51.295,-47.838,179.522,5.375,149.081
C06127=1126.696,-51.544,-47.827,179.523,5.371,149.080
C06128=1126.701,-51.795,-47.817,179.523,5.366,149.079
C06129=1126.706,-52.044,-47.806,179.523,5.362,149.078
C06130=1126.711,-52.294,-47.795,179.523,5.357,149.077
C06131=1126.717,-52.543,-47.785,179.524,5.353,149.075
C06132=1126.722,-52.793,-47.774,179.524,5.348,149.075
C06133=1126.727,-53.043,-47.763,179.524,5.343,149.073
C06134=1126.732,-53.293,-47.753,179.524,5.338,149.072
C06135=1126.737,-53.542,-47.742,179.524,5.334,149.071
C06136=1126.743,-53.791,-47.732,179.525,5.329,149.070
C06137=1126.749,-54.042,-47.721,179.525,5.324,149.069
C06138=1126.754,-54.291,-47.710,179.525,5.320,149.068
C06139=1126.759,-54.541,-47.699,179.525,5.315,149.067
C06140=1126.765,-54.791,-47.689,179.525,5.310,149.066
C06141=1126.770,-55.041,-47.678,179.525,5.306,149.065
C06142=1126.775,-55.290,-47.667,179.525,5.301,149.064
C06143=1126.780,-55.540,-47.657,179.526,5.296,149.063
C06144=1126.786,-55.790,-47.647,179.526,5.292,149.062
C06145=1126.791,-56.040,-47.636,179.526,5.287,149.061
C06146=1126.796,-56.289,-47.626,179.526,5.282,149.059
C06147=1126.801,-56.538,-47.615,179.527,5.278,149.059
C06148=1126.806,-56.788,-47.604,179.527,5.273,149.057
C06149=1126.812,-57.038,-47.594,179.527,5.269,149.056
C06150=1126.817,-57.288,-47.583,179.527,5.264,149.055
C06151=1126.823,-57.538,-47.573,179.527,5.259,149.054
C06152=1126.827,-57.787,-47.562,179.528,5.254,149.053
C06153=1126.833,-58.037,-47.552,179.527,5.250,149.052
C06154=1126.839,-58.287,-47.542,179.528,5.245,149.051
C06155=1126.844,-58.537,-47.531,179.528,5.240,149.050
C06156=1126.849,-58.786,-47.521,179.528,5.236,149.049
C06157=1126.854,-59.037,-47.510,179.529,5.231,149.048
C06158=1126.859,-59.285,-47.499,179.529,5.227,149.047
C06159=1126.865,-59.535,-47.489,179.529,5.222,149.046
C06160=1126.870,-59.785,-47.478,179.530,5.218,149.044
C06161=1126.876,-60.035,-47.468,179.529,5.213,149.044
C06162=1126.880,-60.285,-47.458,179.530,5.208,149.042
C06163=1126.885,-60.500,-47.449,179.528,5.203,149.042
C06164=1126.889,-60.716,-47.440,179.528,5.198,149.041
C06165=1126.894,-60.932,-47.431,179.527,5.194,149.040
C06166=1126.899,-61.147,-47.422,179.526,5.190,149.039
C06167=1126.903,-61.363,-47.414,179.526,5.185,149.039
C06168=1126.908,-61.579,-47.405,179.525,5.181,149.038
C06169=1126.912,-61.794,-47.395,179.524,5.176,149.037
C06170=1126.917,-62.010,-47.387,179.524,5.171,149.036
C06171=1126.923,-62.260,-47.376,179.522,5.166,149.036
C06172=1126.928,-62.509,-47.367,179.521,5.161,149.035
C06173=1126.933,-62.759,-47.356,179.520,5.155,149.034
C06174=1126.938,-63.009,-47.346,179.520,5.150,149.033
C06175=1126.944,-63.258,-47.336,179.519,5.145,149.032
C06176=1126.949,-63.509,-47.325,179.518,5.139,149.031
C06177=1126.954,-63.758,-47.315,179.517,5.134,149.030
C06178=1126.959,-64.007,-47.305,179.516,5.129,149.029
C06179=1126.964,-64.258,-47.295,179.516,5.123,149.028
C06180=1126.970,-64.507,-47.285,179.515,5.117,149.027
C06181=1126.976,-64.757,-47.275,179.515,5.113,149.026
C06182=1126.981,-65.006,-47.264,179.514,5.107,149.025
C06183=1126.986,-65.257,-47.255,179.513,5.101,149.024
C06184=1126.991,-65.506,-47.245,179.512,5.097,149.023
C06185=1126.997,-65.756,-47.235,179.511,5.091,149.023
C06186=1127.002,-66.005,-47.224,179.511,5.085,149.021
C06187=1127.007,-66.256,-47.214,179.510,5.080,149.021
C06188=1127.012,-66.505,-47.204,179.509,5.075,149.020
C06189=1127.018,-66.755,-47.195,179.509,5.070,149.019
C06190=1127.024,-67.005,-47.185,179.509,5.064,149.018
C06191=1127.028,-67.255,-47.175,179.508,5.059,149.017
C06192=1127.034,-67.504,-47.164,179.507,5.054,149.016
C06193=1127.039,-67.754,-47.154,179.506,5.048,149.015
C06194=1127.045,-68.004,-47.145,179.506,5.043,149.014
C06195=1127.050,-68.253,-47.135,179.505,5.038,149.013
C06196=1127.055,-68.503,-47.124,179.506,5.032,149.012
C06197=1127.061,-68.753,-47.114,179.505,5.027,149.011
C06198=1127.066,-69.003,-47.105,179.504,5.022,149.010
C06199=1127.071,-69.252,-47.095,179.504,5.016,149.009
C06200=1127.077,-69.502,-47.085,179.503,5.011,149.008
C06201=1127.082,-69.752,-47.076,179.503,5.005,149.007
C06202=1127.087,-70.002,-47.065,179.503,5.001,149.006
C06203=1127.093,-70.251,-47.055,179.502,4.995,149.004
C06204=1127.098,-70.501,-47.046,179.502,4.990,149.004
C06205=1127.104,-70.751,-47.036,179.501,4.984,149.002
C06206=1127.108,-71.000,-47.027,179.501,4.979,149.001
C06207=1127.114,-71.250,-47.017,179.501,4.974,149.000
C06208=1127.120,-71.500,-47.007,179.500,4.968,148.999
C06209=1127.124,-71.750,-46.998,179.500,4.963,148.998
C06210=1127.130,-72.000,-46.987,179.500,4.957,148.997
C06211=1127.135,-72.249,-46.978,179.499,4.952,148.996
C06212=1127.141,-72.499,-46.968,179.500,4.947,148.995
C06213=1127.146,-72.749,-46.958,179.499,4.942,148.994
C06214=1127.152,-72.999,-46.949,179.499,4.937,148.993
C06215=1127.157,-73.248,-46.939,179.499,4.931,148.992
C06216=1127.162,-73.498,-46.930,179.498,4.926,148.991
C06217=1127.168,-73.748,-46.920,179.498,4.921,148.990
C06218=1127.173,-73.997,-46.911,179.498,4.916,148.989
C06219=1127.180,-74.313,-46.898,179.498,4.908,148.987
C06220=1127.187,-74.627,-46.886,179.498,4.902,148.986
C06221=1127.193,-74.942,-46.874,179.497,4.895,148.984
C06222=1127.201,-75.257,-46.862,179.497,4.888,148.983
C06223=1127.205,-75.506,-46.853,179.497,4.884,148.982
C06224=1127.211,-75.756,-46.843,179.497,4.879,148.981
C06225=1127.216,-76.006,-46.833,179.497,4.873,148.980
C06226=1127.222,-76.256,-46.824,179.497,4.867,148.979
C06227=1127.227,-76.505,-46.814,179.497,4.862,148.977
C06228=1127.233,-76.755,-46.805,179.497,4.857,148.976
C06229=1127.238,-77.005,-46.796,179.497,4.852,148.975
C06230=1127.243,-77.254,-46.786,179.496,4.846,148.974
C06231=1127.249,-77.504,-46.777,179.496,4.841,148.973
C06232=1127.254,-77.754,-46.767,179.497,4.836,148.972
C06233=1127.260,-78.004,-46.758,179.497,4.831,148.971
C06234=1127.265,-78.254,-46.749,179.497,4.826,148.969
C06235=1127.270,-78.503,-46.739,179.497,4.821,148.968
C06236=1127.275,-78.753,-46.730,179.497,4.815,148.967
C06237=1127.281,-79.003,-46.721,179.497,4.810,148.966
C06238=1127.286,-79.253,-46.711,179.498,4.805,148.965
C06239=1127.291,-79.502,-46.702,179.498,4.800,148.964
C06240=1127.297,-79.753,-46.692,179.497,4.795,148.963
C06241=1127.302,-80.002,-46.683,179.498,4.790,148.962
C06242=1127.307,-80.252,-46.674,179.498,4.785,148.960
C06243=1127.313,-80.502,-46.664,179.498,4.780,148.959
C06244=1127.318,-80.752,-46.655,179.498,4.774,148.958
C06245=1127.324,-81.001,-46.645,179.498,4.769,148.957
C06246=1127.329,-81.251,-46.636,179.498,4.764,148.956
C06247=1127.334,-81.501,-46.627,179.499,4.759,148.954
C06248=1127.340,-81.751,-46.618,179.499,4.753,148.953
C06249=1127.345,-82.001,-46.609,179.499,4.748,148.952
C06250=1127.350,-82.250,-46.599,179.500,4.743,148.951
C06251=1127.356,-82.500,-46.590,179.500,4.738,148.950
C06252=1127.361,-82.750,-46.581,179.500,4.733,148.948
C06253=1127.367,-82.999,-46.572,179.500,4.728,148.947
C06254=1127.396,-84.346,-46.519,178.735,6.193,149.491
C06255=1127.403,-84.711,-46.505,178.732,6.192,149.492
C06256=1127.409,-84.962,-46.495,178.730,6.192,149.492
C06257=1127.413,-85.211,-46.486,178.728,6.191,149.493
C06258=1127.419,-85.461,-46.476,178.726,6.190,149.493
C06259=1127.424,-85.710,-46.467,178.723,6.189,149.494
C06260=1127.430,-85.960,-46.457,178.722,6.189,149.494
C06261=1127.435,-86.210,-46.448,178.720,6.189,149.495
C06262=1127.440,-86.459,-46.439,178.717,6.188,149.495
C06263=1127.446,-86.710,-46.429,178.715,6.188,149.496
C06264=1127.451,-86.959,-46.420,178.713,6.188,149.497
C06265=1127.457,-87.209,-46.410,178.711,6.187,149.497
C06266=1127.462,-87.459,-46.401,178.709,6.186,149.498
C06267=1127.468,-87.708,-46.391,178.707,6.186,149.498
C06268=1127.473,-87.958,-46.382,178.705,6.185,149.498
C06269=1127.478,-88.208,-46.373,178.703,6.185,149.499
C06270=1127.484,-88.458,-46.363,178.701,6.184,149.499
C06271=1127.489,-88.707,-46.354,178.699,6.184,149.500
C06272=1127.495,-88.958,-46.345,178.697,6.183,149.500
C06273=1127.499,-89.207,-46.335,178.695,6.182,149.501
C06274=1127.505,-89.457,-46.326,178.692,6.182,149.501
C06275=1127.511,-89.707,-46.317,178.691,6.182,149.502
C06276=1127.515,-89.956,-46.307,178.689,6.181,149.502
C06277=1127.521,-90.206,-46.298,178.686,6.180,149.503
C06278=1127.526,-90.456,-46.289,178.685,6.180,149.503
C06279=1127.531,-90.705,-46.279,178.683,6.180,149.504
C06280=1127.536,-90.955,-46.270,178.680,6.179,149.504
C06281=1127.542,-91.205,-46.261,178.679,6.179,149.505
C06282=1127.548,-91.455,-46.252,178.676,6.179,149.505
C06283=1127.552,-91.704,-46.242,178.674,6.178,149.506
C06284=1127.558,-91.955,-46.233,178.672,6.177,149.506
C06285=1127.563,-92.204,-46.224,178.670,6.177,149.507
C06286=1127.569,-92.454,-46.215,178.668,6.176,149.507
C06287=1127.574,-92.704,-46.205,178.666,6.176,149.508
C06288=1127.579,-92.954,-46.196,178.664,6.176,149.508
C06289=1127.585,-93.204,-46.187,178.662,6.175,149.509
C06290=1127.591,-93.454,-46.177,178.660,6.174,149.509
C06291=1127.596,-93.702,-46.168,178.658,6.174,149.510
C06292=1127.601,-93.952,-46.159,178.656,6.173,149.510
C06293=1127.607,-94.202,-46.150,178.654,6.173,149.511
C06294=1127.612,-94.452,-46.141,178.652,6.172,149.511
C06295=1127.617,-94.702,-46.132,178.650,6.172,149.512
C06296=1127.622,-94.951,-46.122,178.648,6.171,149.512
C06297=1127.628,-95.201,-46.113,178.646,6.170,149.513
C06298=1127.633,-95.451,-46.104,178.644,6.170,149.513
C06299=1127.638,-95.701,-46.095,178.642,6.170,149.514
C06300=1127.644,-95.951,-46.086,178.640,6.169,149.514
C06301=1127.650,-96.201,-46.077,178.638,6.169,149.515
C06302=1127.655,-96.451,-46.068,178.636,6.168,149.515
C06303=1127.660,-96.699,-46.058,178.634,6.168,149.516
C06304=1127.666,-96.950,-46.049,178.632,6.168,149.516
C06305=1127.671,-97.199,-46.040,178.630,6.167,149.517
C06306=1127.676,-97.449,-46.031,178.628,6.166,149.517
C06307=1127.682,-97.699,-46.022,178.626,6.166,149.518
C06308=1127.687,-97.949,-46.013,178.624,6.165,149.518
C06309=1127.693,-98.199,-46.004,178.622,6.165,149.519
C06310=1127.698,-98.449,-45.995,178.620,6.165,149.519
C06311=1127.703,-98.699,-45.986,178.618,6.164,149.520
C06312=1127.709,-98.948,-45.978,178.616,6.163,149.520
C06313=1127.714,-99.198,-45.967,178.614,6.163,149.521
C06314=1127.720,-99.447,-45.958,178.612,6.163,149.521
C06315=1127.725,-99.697,-45.950,178.610,6.162,149.522
C06316=1127.730,-99.947,-45.941,178.608,6.162,149.522
C06317=1127.735,-100.197,-45.932,178.606,6.161,149.522
C06318=1127.741,-100.447,-45.922,178.604,6.160,149.523
C06319=1127.747,-100.696,-45.914,178.602,6.160,149.523
C06320=1127.752,-100.946,-45.905,178.600,6.160,149.524
C06321=1127.757,-101.196,-45.896,178.598,6.159,149.524
C06322=1127.762,-101.446,-45.887,178.596,6.159,149.525
C06323=1127.767,-101.696,-45.878,178.594,6.158,149.525
C06324=1127.773,-101.946,-45.869,178.592,6.157,149.526
C06325=1127.779,-102.195,-45.860,178.590,6.157,149.526
C06326=1127.784,-102.445,-45.851,178.588,6.157,149.527
C06327=1127.789,-102.695,-45.842,178.586,6.157,149.527
C06328=1127.795,-102.967,-45.833,178.584,6.156,149.528
C06329=1127.801,-103.240,-45.823,178.581,6.156,149.529
C06330=1127.807,-103.512,-45.814,178.579,6.155,149.529
C06331=1127.812,-103.784,-45.804,178.577,6.154,149.530
C06332=1127.818,-104.033,-45.795,178.575,6.154,149.530
C06333=1127.823,-104.283,-45.786,178.573,6.154,149.531
C06334=1127.829,-104.534,-45.778,178.572,6.154,149.531
C06335=1127.834,-104.784,-45.769,178.569,6.153,149.531
C06336=1127.839,-105.033,-45.760,178.567,6.152,149.532
C06337=1127.845,-105.283,-45.751,178.566,6.152,149.532
C06338=1127.851,-105.533,-45.742,178.563,6.151,149.533
C06339=1127.856,-105.783,-45.733,178.561,6.151,149.533
C06340=1127.861,-106.032,-45.724,178.560,6.151,149.534
C06341=1127.866,-106.282,-45.715,178.557,6.150,149.534
C06342=1127.872,-106.531,-45.707,178.555,6.149,149.535
C06343=1127.877,-106.781,-45.698,178.554,6.149,149.535
C06344=1127.883,-107.032,-45.690,178.551,6.148,149.536
C06345=1127.888,-107.282,-45.681,178.550,6.149,149.536
C06346=1127.893,-107.531,-45.672,178.548,6.148,149.537
C06347=1127.899,-107.781,-45.663,178.546,6.147,149.537
C06348=1127.904,-108.031,-45.655,178.544,6.147,149.538
C06349=1127.909,-108.280,-45.646,178.542,6.146,149.538
C06350=1127.915,-108.530,-45.638,178.541,6.146,149.539
C06351=1127.920,-108.780,-45.629,178.538,6.145,149.539
C06352=1127.925,-109.030,-45.620,178.536,6.145,149.540
C06353=1127.931,-109.280,-45.611,178.535,6.145,149.540
C06354=1127.936,-109.529,-45.603,178.532,6.144,149.540
C06355=1127.942,-109.779,-45.594,178.531,6.144,149.541
C06356=1127.947,-110.029,-45.586,178.529,6.143,149.541
C06357=1127.952,-110.279,-45.577,178.526,6.142,149.542
C06358=1127.958,-110.528,-45.568,178.525,6.142,149.542
C06359=1127.963,-110.778,-45.559,178.523,6.142,149.543
C06360=1127.969,-111.028,-45.551,178.521,6.142,149.543
C06361=1127.974,-111.278,-45.543,178.519,6.141,149.544
C06362=1127.979,-111.527,-45.534,178.517,6.140,149.544
C06363=1127.985,-111.777,-45.525,178.515,6.140,149.545
C06364=1127.990,-112.028,-45.517,178.513,6.140,149.545
C06365=1127.996,-112.277,-45.508,178.511,6.140,149.546
C06366=1128.001,-112.527,-45.499,178.509,6.139,149.546
C06367=1128.007,-112.777,-45.491,178.507,6.138,149.547
C06368=1128.012,-113.026,-45.482,178.506,6.138,149.547
C06369=1128.017,-113.276,-45.474,178.504,6.137,149.548
C06370=1128.023,-113.526,-45.465,178.502,6.137,149.548
C06371=1128.028,-113.776,-45.457,178.500,6.136,149.549
C06372=1128.033,-114.025,-45.448,178.498,6.136,149.549
C06373=1128.038,-114.275,-45.440,178.496,6.136,149.550
C06374=1128.044,-114.525,-45.432,178.494,6.135,149.550
C06375=1128.050,-114.775,-45.423,178.492,6.135,149.550
C06376=1128.055,-115.025,-45.414,178.490,6.134,149.551
C06377=1128.061,-115.275,-45.406,178.488,6.134,149.551
C06378=1128.066,-115.524,-45.397,178.486,6.134,149.552
C06379=1128.071,-115.774,-45.388,178.484,6.133,149.552
C06380=1128.077,-116.024,-45.381,178.482,6.133,149.553
C06381=1128.082,-116.274,-45.372,178.481,6.132,149.553
C06382=1128.087,-116.524,-45.364,178.479,6.132,149.554
C06383=1128.093,-116.773,-45.356,178.477,6.131,149.554
C06384=1128.098,-117.023,-45.347,178.475,6.131,149.555
C06385=1128.104,-117.273,-45.339,178.473,6.130,149.555
C06386=1128.109,-117.523,-45.330,178.471,6.130,149.556
C06387=1128.115,-117.773,-45.322,178.469,6.130,149.556
C06388=1128.120,-118.022,-45.313,178.467,6.129,149.557
C06389=1128.125,-118.272,-45.305,178.465,6.129,149.557
C06390=1128.130,-118.522,-45.297,178.463,6.128,149.558
C06391=1128.136,-118.771,-45.288,178.462,6.128,149.558
C06392=1128.142,-119.022,-45.280,178.460,6.127,149.558
C06393=1128.147,-119.271,-45.271,178.458,6.126,149.559
C06394=1128.153,-119.522,-45.263,178.456,6.126,149.559
C06395=1128.157,-119.771,-45.255,178.454,6.126,149.560
C06396=1128.163,-120.021,-45.247,178.452,6.126,149.560
C06397=1128.169,-120.271,-45.238,178.450,6.125,149.561
C06398=1128.174,-120.521,-45.229,178.449,6.125,149.561
C06399=1128.180,-120.770,-45.222,178.446,6.124,149.562
C06400=1128.184,-121.020,-45.213,178.445,6.124,149.562
C06401=1128.190,-121.270,-45.205,178.443,6.124,149.563
C06402=1128.195,-121.519,-45.197,178.441,6.123,149.563
C06403=1128.202,-121.769,-45.189,178.439,6.123,149.563
C06404=1128.206,-122.019,-45.180,178.437,6.122,149.564
C06405=1128.211,-122.269,-45.172,178.435,6.122,149.564
C06406=1128.217,-122.519,-45.164,178.433,6.121,149.565
C06407=1128.223,-122.769,-45.156,178.432,6.121,149.565
C06408=1128.229,-123.019,-45.148,178.429,6.120,149.566
C06409=1128.233,-123.268,-45.139,178.428,6.120,149.566
C06410=1128.239,-123.519,-45.131,178.426,6.119,149.567
C06411=1128.244,-123.768,-45.123,178.425,6.119,149.567
C06412=1128.250,-124.018,-45.115,178.422,6.119,149.568
C06413=1128.255,-124.267,-45.107,178.421,6.119,149.568
C06414=1128.260,-124.518,-45.098,178.419,6.118,149.569
C06415=1128.266,-124.767,-45.091,178.416,6.117,149.569
C06416=1128.271,-125.017,-45.082,178.415,6.117,149.570
C06417=1128.277,-125.267,-45.074,178.413,6.117,149.570
C06418=1128.282,-125.516,-45.066,178.411,6.116,149.570
C06419=1128.288,-125.766,-45.058,178.409,6.115,149.571
C06420=1128.293,-126.016,-45.050,178.408,6.116,149.571
C06421=1128.298,-126.266,-45.041,178.405,6.115,149.572
C06422=1128.304,-126.516,-45.033,178.404,6.115,149.572
C06423=1128.309,-126.766,-45.025,178.402,6.114,149.573
C06424=1128.315,-127.015,-45.017,178.400,6.114,149.573
C06425=1128.320,-127.266,-45.009,178.398,6.113,149.574
C06426=1128.325,-127.515,-45.001,178.397,6.113,149.574
C06427=1128.331,-127.765,-44.993,178.395,6.112,149.575
C06428=1128.337,-128.015,-44.985,178.393,6.112,149.575
C06429=1128.341,-128.264,-44.977,178.391,6.112,149.575
C06430=1128.347,-128.514,-44.969,178.389,6.112,149.576
C06431=1128.353,-128.765,-44.961,178.387,6.111,149.576
C06432=1127.932,-128.775,-45.005,178.384,6.115,149.578
C06433=1127.926,-128.525,-45.013,178.386,6.115,149.578
C06434=1127.921,-128.275,-45.022,178.388,6.115,149.577
C06435=1127.916,-128.026,-45.029,178.389,6.116,149.577
C06436=1127.910,-127.776,-45.038,178.391,6.116,149.576
C06437=1127.904,-127.526,-45.046,178.393,6.116,149.576
C06438=1127.900,-127.276,-45.054,178.395,6.117,149.575
C06439=1127.894,-127.026,-45.061,178.397,6.117,149.575
C06440=1127.888,-126.777,-45.070,178.399,6.118,149.574
C06441=1127.883,-126.527,-45.078,178.400,6.118,149.574
C06442=1127.878,-126.277,-45.086,178.402,6.119,149.574
C06443=1127.872,-126.028,-45.094,178.404,6.119,149.573
C06444=1127.867,-125.777,-45.102,178.406,6.120,149.573
C06445=1127.861,-125.528,-45.110,178.408,6.120,149.572
C06446=1127.856,-125.278,-45.119,178.410,6.120,149.572
C06447=1127.850,-125.029,-45.127,178.412,6.121,149.571
C06448=1127.845,-124.778,-45.135,178.414,6.121,149.571
C06449=1127.839,-124.529,-45.143,178.415,6.122,149.570
C06450=1127.834,-124.279,-45.151,178.417,6.122,149.570
C06451=1127.829,-124.029,-45.159,178.419,6.123,149.569
C06452=1127.824,-123.780,-45.168,178.421,6.123,149.569
C06453=1127.818,-123.529,-45.176,178.423,6.123,149.568
C06454=1127.812,-123.280,-45.184,178.425,6.123,149.568
C06455=1127.808,-123.030,-45.192,178.427,6.124,149.567
C06456=1127.802,-122.780,-45.200,178.428,6.124,149.567
C06457=1127.796,-122.530,-45.209,178.430,6.125,149.567
C06458=1127.790,-122.280,-45.216,178.432,6.125,149.566
C06459=1127.786,-122.031,-45.225,178.434,6.126,149.566
C06460=1127.780,-121.780,-45.233,178.436,6.127,149.565
C06461=1127.775,-121.531,-45.241,178.438,6.127,149.565
C06462=1127.769,-121.281,-45.250,178.440,6.127,149.564
C06463=1127.763,-121.032,-45.258,178.441,6.127,149.564
C06464=1127.759,-120.781,-45.266,178.444,6.128,149.563
C06465=1127.754,-120.532,-45.275,178.445,6.128,149.563
C06466=1127.747,-120.282,-45.282,178.447,6.129,149.563
C06467=1127.742,-120.032,-45.291,178.449,6.129,149.562
C06468=1127.736,-119.782,-45.299,178.451,6.130,149.562
C06469=1127.732,-119.533,-45.307,178.453,6.131,149.561
C06470=1127.727,-119.283,-45.316,178.455,6.130,149.561
C06471=1127.721,-119.033,-45.324,178.457,6.131,149.560
C06472=1127.715,-118.783,-45.333,178.458,6.131,149.560
C06473=1127.709,-118.533,-45.341,178.461,6.132,149.559
C06474=1127.705,-118.284,-45.349,178.462,6.132,149.559
C06475=1127.699,-118.033,-45.357,178.464,6.133,149.558
C06476=1127.694,-117.784,-45.366,178.465,6.133,149.558
C06477=1127.688,-117.534,-45.375,178.468,6.134,149.557
C06478=1127.683,-117.284,-45.383,178.470,6.134,149.557
C06479=1127.677,-117.035,-45.391,178.471,6.134,149.556
C06480=1127.672,-116.784,-45.400,178.474,6.135,149.556
C06481=1127.667,-116.534,-45.409,178.475,6.135,149.555
C06482=1127.662,-116.286,-45.417,178.477,6.136,149.555
C06483=1127.656,-116.035,-45.425,178.479,6.136,149.555
C06484=1127.650,-115.786,-45.433,178.481,6.136,149.554
C06485=1127.645,-115.535,-45.441,178.483,6.138,149.554
C06486=1127.640,-115.286,-45.450,178.485,6.138,149.553
C06487=1127.634,-115.036,-45.459,178.487,6.138,149.553
C06488=1127.628,-114.786,-45.467,178.488,6.138,149.552
C06489=1127.623,-114.536,-45.476,178.491,6.139,149.552
C06490=1127.618,-114.287,-45.484,178.492,6.139,149.551
C06491=1127.613,-114.037,-45.492,178.494,6.140,149.551
C06492=1127.608,-113.787,-45.501,178.497,6.140,149.550
C06493=1127.602,-113.538,-45.509,178.498,6.140,149.550
C06494=1127.596,-113.287,-45.518,178.500,6.141,149.549
C06495=1127.591,-113.038,-45.527,178.502,6.141,149.549
C06496=1127.585,-112.788,-45.535,178.504,6.142,149.548
C06497=1127.580,-112.539,-45.544,178.506,6.143,149.548
C06498=1127.575,-112.288,-45.552,178.507,6.143,149.548
C06499=1127.570,-112.038,-45.561,178.510,6.144,149.547
C06500=1127.564,-111.789,-45.570,178.511,6.144,149.547
C06501=1127.558,-111.539,-45.578,178.513,6.144,149.546
C06502=1127.553,-111.289,-45.587,178.516,6.145,149.546
C06503=1127.547,-111.040,-45.595,178.517,6.145,149.545
C06504=1127.542,-110.790,-45.604,178.519,6.146,149.545
C06505=1127.537,-110.539,-45.612,178.521,6.146,149.544
C06506=1127.532,-110.289,-45.621,178.523,6.146,149.544
C06507=1127.526,-110.040,-45.630,178.525,6.147,149.543
C06508=1127.521,-109.790,-45.639,178.527,6.147,149.543
C06509=1127.516,-109.541,-45.648,178.529,6.148,149.542
C06510=1127.509,-109.291,-45.655,178.531,6.148,149.542
C06511=1127.504,-109.041,-45.664,178.533,6.149,149.541
C06512=1127.499,-108.791,-45.673,178.535,6.149,149.541
C06513=1127.494,-108.541,-45.682,178.537,6.149,149.540
C06514=1127.488,-108.292,-45.691,178.539,6.150,149.540
C06515=1127.483,-108.042,-45.699,178.541,6.150,149.539
C06516=1127.478,-107.792,-45.708,178.543,6.151,149.539
C06517=1127.472,-107.542,-45.717,178.545,6.152,149.539
C06518=1127.467,-107.293,-45.725,178.546,6.152,149.538
C06519=1127.461,-107.043,-45.734,178.548,6.153,149.538
C06520=1127.456,-106.793,-45.743,178.550,6.153,149.537
C06521=1127.451,-106.543,-45.752,178.552,6.153,149.537
C06522=1127.446,-106.293,-45.760,178.554,6.154,149.536
C06523=1127.440,-106.044,-45.768,178.556,6.154,149.536
C06524=1127.435,-105.794,-45.777,178.558,6.155,149.535
C06525=1127.430,-105.544,-45.786,178.560,6.155,149.535
C06526=1127.424,-105.294,-45.795,178.562,6.155,149.534
C06527=1127.419,-105.045,-45.804,178.564,6.156,149.534
C06528=1127.413,-104.795,-45.813,178.566,6.157,149.533
C06529=1127.408,-104.545,-45.821,178.568,6.157,149.533
C06530=1127.402,-104.295,-45.831,178.570,6.158,149.532
C06531=1127.397,-104.045,-45.840,178.572,6.158,149.532
C06532=1127.391,-103.795,-45.848,178.574,6.158,149.531
C06533=1127.386,-103.523,-45.858,178.576,6.159,149.531
C06534=1127.380,-103.251,-45.867,178.578,6.160,149.530
C06535=1127.374,-102.978,-45.877,178.580,6.160,149.530
C06536=1127.368,-102.706,-45.886,178.583,6.160,149.529
C06537=1127.363,-102.456,-45.895,178.585,6.161,149.529
C06538=1127.358,-102.206,-45.904,178.586,6.161,149.528
C06539=1127.352,-101.957,-45.913,178.589,6.161,149.528
C06540=1127.347,-101.707,-45.922,178.591,6.162,149.527
C06541=1127.341,-101.457,-45.931,178.592,6.162,149.527
C06542=1127.336,-101.207,-45.940,178.595,6.163,149.526
C06543=1127.331,-100.957,-45.949,178.597,6.164,149.526
C06544=1127.326,-100.707,-45.958,178.598,6.164,149.525
C06545=1127.320,-100.458,-45.966,178.600,6.164,149.525
C06546=1127.315,-100.208,-45.975,178.603,6.165,149.524
C06547=1127.309,-99.958,-45.985,178.604,6.165,149.524
C06548=1127.304,-99.708,-45.994,178.606,6.166,149.523
C06549=1127.298,-99.459,-46.003,178.609,6.167,149.523
C06550=1127.294,-99.209,-46.012,178.610,6.167,149.522
C06551=1127.288,-98.959,-46.021,178.612,6.167,149.522
C06552=1127.282,-98.710,-46.030,178.615,6.168,149.521
C06553=1127.277,-98.460,-46.039,178.616,6.168,149.521
C06554=1127.272,-98.210,-46.048,178.618,6.169,149.520
C06555=1127.266,-97.960,-46.057,178.621,6.169,149.520
C06556=1127.261,-97.711,-46.066,178.622,6.169,149.519
C06557=1127.255,-97.460,-46.075,178.624,6.170,149.519
C06558=1127.250,-97.211,-46.084,178.627,6.171,149.518
C06559=1127.245,-96.961,-46.093,178.628,6.171,149.518
C06560=1127.239,-96.712,-46.102,178.630,6.172,149.517
C06561=1127.234,-96.462,-46.112,178.633,6.172,149.517
C06562=1127.228,-96.212,-46.121,178.634,6.172,149.517
C06563=1127.223,-95.962,-46.130,178.636,6.173,149.516
C06564=1127.218,-95.712,-46.139,178.639,6.174,149.516
C06565=1127.212,-95.462,-46.148,178.640,6.174,149.515
C06566=1127.207,-95.212,-46.157,178.642,6.175,149.515
C06567=1127.202,-94.963,-46.166,178.645,6.175,149.514
C06568=1127.196,-94.713,-46.176,178.646,6.175,149.514
C06569=1127.191,-94.463,-46.185,178.648,6.176,149.513
C06570=1127.186,-94.213,-46.194,178.651,6.177,149.513
C06571=1127.181,-93.964,-46.203,178.653,6.177,149.512
C06572=1127.174,-93.714,-46.212,178.654,6.177,149.512
C06573=1127.150,-92.530,-46.259,179.527,4.544,148.899
C06574=1127.144,-92.280,-46.268,179.526,4.548,148.901
C06575=1127.139,-92.030,-46.277,179.525,4.553,148.902
C06576=1127.134,-91.781,-46.285,179.525,4.558,148.903
C06577=1127.128,-91.531,-46.294,179.524,4.563,148.904
C06578=1127.122,-91.281,-46.303,179.523,4.567,148.906
C06579=1127.117,-91.031,-46.312,179.523,4.572,148.907
C06580=1127.112,-90.782,-46.321,179.521,4.577,148.908
C06581=1127.107,-90.532,-46.330,179.521,4.582,148.909
C06582=1127.102,-90.282,-46.339,179.520,4.586,148.911
C06583=1127.096,-90.033,-46.348,179.520,4.592,148.912
C06584=1127.090,-89.783,-46.357,179.519,4.596,148.913
C06585=1127.085,-89.533,-46.366,179.519,4.602,148.914
C06586=1127.081,-89.304,-46.374,179.518,4.606,148.916
C06587=1127.076,-89.075,-46.382,179.518,4.610,148.916
C06588=1127.070,-88.847,-46.391,179.517,4.614,148.918
C06589=1127.065,-88.618,-46.399,179.517,4.619,148.919
C06590=1127.061,-88.390,-46.407,179.516,4.624,148.920
C06591=1127.056,-88.161,-46.416,179.516,4.628,148.921
C06592=1127.051,-87.932,-46.424,179.515,4.632,148.922
C06593=1127.045,-87.704,-46.432,179.515,4.637,148.923
C06594=1127.040,-87.454,-46.441,179.514,4.642,148.924
C06595=1127.035,-87.205,-46.450,179.514,4.647,148.926
C06596=1127.030,-86.955,-46.459,179.513,4.652,148.927
C06597=1127.025,-86.705,-46.468,179.512,4.657,148.928
C06598=1127.019,-86.455,-46.477,179.512,4.662,148.929
C06599=1127.014,-86.205,-46.486,179.512,4.667,148.931
C06600=1127.008,-85.955,-46.495,179.511,4.671,148.932
C06601=1127.003,-85.705,-46.504,179.510,4.677,148.933
C06602=1126.997,-85.456,-46.514,179.510,4.682,148.934
C06603=1126.992,-85.206,-46.523,179.510,4.687,148.936
C06604=1126.987,-84.957,-46.532,179.509,4.692,148.937
C06605=1126.982,-84.707,-46.541,179.509,4.697,148.938
C06606=1126.976,-84.457,-46.550,179.509,4.702,148.939
C06607=1126.970,-84.207,-46.559,179.509,4.707,148.940
C06608=1126.966,-83.958,-46.569,179.508,4.711,148.941
C06609=1126.960,-83.707,-46.578,179.507,4.717,148.943
C06610=1126.955,-83.458,-46.587,179.507,4.722,148.944
C06611=1126.949,-83.208,-46.596,179.507,4.727,148.945
C06612=1126.943,-82.957,-46.605,179.507,4.733,148.946
C06613=1126.939,-82.708,-46.615,179.507,4.738,148.947
C06614=1126.933,-82.458,-46.624,179.506,4.743,148.949
C06615=1126.927,-82.209,-46.633,179.506,4.748,148.950
C06616=1126.922,-81.959,-46.642,179.505,4.752,148.951
C06617=1126.917,-81.710,-46.652,179.505,4.758,148.952
C06618=1126.911,-81.460,-46.661,179.505,4.763,148.953
C06619=1126.906,-81.210,-46.670,179.505,4.768,148.954
C06620=1126.901,-80.960,-46.679,179.505,4.773,148.956
C06621=1126.895,-80.710,-46.689,179.505,4.778,148.957
C06622=1126.890,-80.461,-46.698,179.505,4.783,148.958
C06623=1126.885,-80.211,-46.707,179.504,4.789,148.959
C06624=1126.879,-79.961,-46.717,179.504,4.794,148.960
C06625=1126.874,-79.711,-46.726,179.504,4.799,148.961
C06626=1126.868,-79.461,-46.735,179.504,4.804,148.963
C06627=1126.863,-79.212,-46.745,179.504,4.809,148.964
C06628=1126.857,-78.962,-46.755,179.504,4.814,148.965
C06629=1126.852,-78.712,-46.763,179.503,4.819,148.966
C06630=1126.847,-78.463,-46.773,179.504,4.825,148.967
C06631=1126.841,-78.213,-46.783,179.504,4.831,148.968
C06632=1126.836,-77.963,-46.791,179.503,4.836,148.970
C06633=1126.831,-77.713,-46.802,179.503,4.841,148.971
C06634=1126.825,-77.463,-46.811,179.503,4.846,148.972
C06635=1126.820,-77.214,-46.821,179.503,4.851,148.973
C06636=1126.815,-76.964,-46.830,179.503,4.856,148.974
C06637=1126.809,-76.714,-46.839,179.503,4.861,148.975
C06638=1126.804,-76.465,-46.849,179.504,4.867,148.976
C06639=1126.798,-76.214,-46.858,179.504,4.872,148.978
C06640=1126.793,-75.965,-46.868,179.503,4.877,148.979
C06641=1126.787,-75.715,-46.877,179.503,4.883,148.980
C06642=1126.783,-75.499,-46.885,179.504,4.887,148.981
C06643=1126.778,-75.283,-46.894,179.504,4.892,148.982
C06644=1126.774,-75.068,-46.903,179.504,4.896,148.983
C06645=1126.770,-74.852,-46.911,179.504,4.901,148.984
C06646=1126.764,-74.637,-46.919,179.504,4.906,148.984
C06647=1126.760,-74.421,-46.927,179.504,4.910,148.985
C06648=1126.755,-74.205,-46.935,179.505,4.914,148.986
C06649=1126.751,-73.989,-46.943,179.505,4.919,148.987
C06650=1126.745,-73.739,-46.954,179.505,4.924,148.988
C06651=1126.740,-73.490,-46.962,179.505,4.930,148.990
C06652=1126.735,-73.240,-46.973,179.505,4.935,148.991
C06653=1126.729,-72.990,-46.982,179.505,4.940,148.992
C06654=1126.724,-72.741,-46.992,179.505,4.945,148.993
C06655=1126.718,-72.491,-47.002,179.506,4.951,148.994
C06656=1126.714,-72.240,-47.011,179.506,4.956,148.995
C06657=1126.708,-71.991,-47.021,179.506,4.961,148.996
C06658=1126.702,-71.741,-47.031,179.507,4.967,148.997
C06659=1126.697,-71.492,-47.041,179.507,4.972,148.998
C06660=1126.692,-71.242,-47.051,179.508,4.978,148.999
C06661=1126.687,-70.992,-47.060,179.508,4.983,149.000
C06662=1126.681,-70.743,-47.070,179.507,4.988,149.001
C06663=1126.676,-70.492,-47.080,179.508,4.994,149.002
C06664=1126.671,-70.243,-47.089,179.508,4.999,149.003
C06665=1126.665,-69.993,-47.100,179.509,5.004,149.004
C06666=1126.660,-69.743,-47.110,179.509,5.009,149.006
C06667=1126.654,-69.494,-47.119,179.510,5.015,149.006
C06668=1126.649,-69.244,-47.129,179.510,5.020,149.008
C06669=1126.644,-68.994,-47.139,179.511,5.026,149.009
C06670=1126.639,-68.745,-47.149,179.511,5.030,149.009
C06671=1126.633,-68.494,-47.159,179.512,5.036,149.011
C06672=1126.627,-68.245,-47.169,179.512,5.041,149.011
C06673=1126.622,-67.995,-47.179,179.513,5.047,149.013
C06674=1126.618,-67.745,-47.189,179.513,5.052,149.014
C06675=1126.612,-67.495,-47.198,179.514,5.057,149.014
C06676=1126.606,-67.246,-47.209,179.514,5.063,149.016
C06677=1126.601,-66.996,-47.218,179.515,5.068,149.017
C06678=1126.596,-66.746,-47.229,179.515,5.073,149.017
C06679=1126.591,-66.497,-47.239,179.516,5.079,149.018
C06680=1126.585,-66.247,-47.249,179.517,5.085,149.020
C06681=1126.579,-65.997,-47.259,179.517,5.089,149.020
C06682=1126.575,-65.747,-47.269,179.518,5.095,149.021
C06683=1126.569,-65.497,-47.279,179.518,5.100,149.022
C06684=1126.564,-65.248,-47.289,179.519,5.105,149.023
C06685=1126.558,-64.998,-47.299,179.520,5.111,149.024
C06686=1126.554,-64.748,-47.309,179.520,5.116,149.025
C06687=1126.548,-64.499,-47.320,179.521,5.121,149.026
C06688=1126.543,-64.249,-47.330,179.522,5.127,149.027
C06689=1126.537,-64.000,-47.340,179.523,5.132,149.028
C06690=1126.532,-63.750,-47.351,179.523,5.137,149.029
C06691=1126.526,-63.500,-47.361,179.524,5.143,149.030
C06692=1126.521,-63.250,-47.370,179.525,5.148,149.031
C06693=1126.516,-63.000,-47.380,179.526,5.153,149.032
C06694=1126.511,-62.750,-47.390,179.527,5.159,149.033
C06695=1126.505,-62.501,-47.401,179.528,5.164,149.033
C06696=1126.500,-62.251,-47.412,179.528,5.169,149.034
C06697=1126.495,-62.002,-47.422,179.529,5.175,149.035
C06698=1126.490,-61.786,-47.431,179.530,5.179,149.036
C06699=1126.486,-61.570,-47.439,179.530,5.184,149.037
C06700=1126.481,-61.355,-47.449,179.531,5.188,149.038
C06701=1126.476,-61.139,-47.457,179.533,5.193,149.038
C06702=1126.472,-60.923,-47.467,179.533,5.198,149.039
C06703=1126.468,-60.708,-47.475,179.534,5.203,149.040
C06704=1126.463,-60.492,-47.484,179.535,5.207,149.041
C06705=1126.458,-60.276,-47.493,179.535,5.212,149.041
C06706=1126.453,-60.026,-47.504,179.536,5.216,149.042
C06707=1126.448,-59.777,-47.514,179.535,5.221,149.043
C06708=1126.442,-59.527,-47.524,179.535,5.226,149.044
C06709=1126.437,-59.278,-47.535,179.535,5.230,149.046
C06710=1126.432,-59.028,-47.546,179.535,5.235,149.047
C06711=1126.427,-58.778,-47.556,179.534,5.239,149.048
C06712=1126.421,-58.528,-47.566,179.534,5.244,149.049
C06713=1126.416,-58.279,-47.577,179.534,5.249,149.050
C06714=1126.411,-58.028,-47.587,179.534,5.253,149.051
C06715=1126.405,-57.780,-47.598,179.533,5.258,149.052
C06716=1126.400,-57.529,-47.609,179.533,5.263,149.053
C06717=1126.395,-57.280,-47.619,179.533,5.267,149.054
C06718=1126.390,-57.029,-47.629,179.533,5.272,149.055
C06719=1126.384,-56.780,-47.640,179.533,5.277,149.056
C06720=1126.379,-56.530,-47.651,179.533,5.281,149.057
C06721=1126.374,-56.281,-47.661,179.533,5.286,149.058
C06722=1126.368,-56.031,-47.671,179.532,5.290,149.060
C06723=1126.363,-55.781,-47.682,179.532,5.295,149.061
C06724=1126.358,-55.532,-47.693,179.532,5.300,149.062
C06725=1126.353,-55.282,-47.703,179.532,5.305,149.063
C06726=1126.347,-55.032,-47.714,179.531,5.309,149.064
C06727=1126.343,-54.783,-47.725,179.531,5.314,149.065
C06728=1126.337,-54.533,-47.735,179.531,5.319,149.066
C06729=1126.332,-54.283,-47.746,179.531,5.323,149.067
C06730=1126.326,-54.033,-47.756,179.531,5.328,149.068
C06731=1126.321,-53.783,-47.768,179.530,5.332,149.069
C06732=1126.315,-53.534,-47.778,179.531,5.337,149.070
C06733=1126.310,-53.284,-47.789,179.530,5.342,149.071
C06734=1126.305,-53.035,-47.799,179.530,5.347,149.072
C06735=1126.300,-52.784,-47.810,179.530,5.351,149.073
C06736=1126.294,-52.535,-47.820,179.530,5.356,149.074
C06737=1126.290,-52.285,-47.832,179.529,5.361,149.076
C06738=1126.284,-52.036,-47.842,179.529,5.365,149.077
C06739=1126.279,-51.785,-47.852,179.529,5.370,149.078
C06740=1126.273,-51.536,-47.864,179.529,5.374,149.079
C06741=1126.268,-51.286,-47.874,179.528,5.380,149.080
C06742=1126.263,-51.037,-47.885,179.528,5.383,149.081
C06743=1126.258,-50.787,-47.896,179.528,5.389,149.082
C06744=1126.252,-50.537,-47.906,179.528,5.394,149.083
C06745=1126.248,-50.288,-47.917,179.528,5.398,149.084
C06746=1126.241,-50.038,-47.928,179.528,5.403,149.085
C06747=1126.237,-49.788,-47.940,179.527,5.407,149.086
C06748=1126.231,-49.539,-47.950,179.528,5.412,149.087
C06749=1126.226,-49.289,-47.961,179.527,5.416,149.088
C06750=1126.221,-49.039,-47.971,179.527,5.421,149.090
C06751=1126.215,-48.789,-47.982,179.527,5.427,149.091
C06752=1126.210,-48.540,-47.993,179.527,5.431,149.092
C06753=1126.205,-48.290,-48.004,179.527,5.436,149.093
C06754=1126.200,-48.074,-48.013,179.526,5.440,149.094
C06755=1126.195,-47.859,-48.022,179.526,5.444,149.095
C06756=1126.191,-47.644,-48.032,179.526,5.448,149.096
C06757=1126.187,-47.428,-48.042,179.526,5.452,149.096
C06758=1126.182,-47.212,-48.051,179.526,5.455,149.097
C06759=1126.178,-46.997,-48.061,179.525,5.459,149.098
C06760=1126.173,-46.781,-48.070,179.525,5.464,149.099
C06761=1126.168,-46.566,-48.079,179.525,5.468,149.100
C06762=1126.164,-46.316,-48.091,179.525,5.472,149.101
C06763=1126.157,-46.066,-48.101,179.525,5.478,149.102
C06764=1126.153,-45.817,-48.113,179.524,5.482,149.104
C06765=1126.147,-45.567,-48.123,179.524,5.487,149.105
C06766=1126.142,-45.317,-48.135,179.524,5.491,149.106
C06767=1126.137,-45.067,-48.145,179.524,5.496,149.107
C06768=1126.131,-44.818,-48.156,179.524,5.501,149.108
C06769=1126.126,-44.568,-48.167,179.524,5.505,149.109
C06770=1126.121,-44.318,-48.179,179.524,5.510,149.110
C06771=1126.116,-44.069,-48.190,179.523,5.515,149.111
C06772=1126.111,-43.819,-48.200,179.523,5.520,149.112
C06773=1126.105,-43.569,-48.212,179.523,5.524,149.113
C06774=1126.100,-43.320,-48.223,179.523,5.529,149.114
C06775=1126.095,-43.069,-48.234,179.523,5.534,149.115
C06776=1126.089,-42.820,-48.245,179.525,5.540,149.116
C06777=1126.084,-42.570,-48.256,179.527,5.546,149.117
C06778=1126.079,-42.320,-48.267,179.529,5.552,149.117
C06779=1126.073,-42.071,-48.279,179.531,5.557,149.118
C06780=1126.068,-41.822,-48.290,179.533,5.563,149.119
C06781=1126.063,-41.571,-48.300,179.534,5.569,149.120
C06782=1126.057,-41.322,-48.312,179.536,5.575,149.120
C06783=1126.053,-41.072,-48.323,179.537,5.580,149.121
C06784=1126.047,-40.822,-48.334,179.540,5.586,149.122
C06785=1126.042,-40.573,-48.345,179.541,5.591,149.122
C06786=1126.037,-40.323,-48.357,179.542,5.596,149.123
C06787=1126.032,-40.073,-48.368,179.544,5.602,149.124
C06788=1126.026,-39.824,-48.379,179.546,5.608,149.124
C06789=1126.021,-39.574,-48.391,179.547,5.613,149.125
C06790=1126.016,-39.324,-48.402,179.548,5.618,149.126
C06791=1126.010,-39.074,-48.414,179.550,5.623,149.127
C06792=1126.005,-38.825,-48.425,179.551,5.629,149.127
C06793=1126.000,-38.575,-48.437,179.552,5.633,149.128
C06794=1125.995,-38.326,-48.448,179.553,5.639,149.129
C06795=1125.990,-38.076,-48.460,179.555,5.644,149.130
C06796=1125.984,-37.827,-48.471,179.556,5.649,149.130
C06797=1125.979,-37.577,-48.483,179.557,5.654,149.131
C06798=1125.974,-37.327,-48.493,179.558,5.659,149.132
C06799=1125.968,-37.077,-48.505,179.559,5.664,149.133
C06800=1125.963,-36.827,-48.517,179.560,5.669,149.134
C06801=1125.958,-36.578,-48.528,179.561,5.673,149.134
C06802=1125.952,-36.328,-48.540,179.561,5.678,149.135
C06803=1125.948,-36.078,-48.551,179.563,5.683,149.136
C06804=1125.942,-35.828,-48.563,179.563,5.688,149.137
C06805=1125.937,-35.579,-48.574,179.564,5.692,149.137
C06806=1125.931,-35.330,-48.586,179.565,5.697,149.138
C06807=1125.926,-35.080,-48.598,179.565,5.702,149.139
C06808=1125.921,-34.830,-48.609,179.566,5.706,149.140
C06809=1125.916,-34.580,-48.621,179.567,5.711,149.141
C06810=1125.912,-34.365,-48.631,179.568,5.715,149.141
C06811=1125.907,-34.149,-48.642,179.568,5.719,149.142
C06812=1125.902,-33.934,-48.651,179.568,5.723,149.143
C06813=1125.898,-33.719,-48.661,179.569,5.727,149.144
C06814=1125.894,-33.503,-48.672,179.569,5.731,149.144
C06815=1125.889,-33.288,-48.681,179.569,5.735,149.145
C06816=1125.885,-33.073,-48.691,179.569,5.738,149.146
C06817=1125.880,-32.857,-48.702,179.570,5.742,149.147
C06818=1125.875,-32.607,-48.714,179.570,5.747,149.147
C06819=1125.870,-32.357,-48.725,179.570,5.751,149.148
C06820=1125.864,-32.108,-48.737,179.570,5.755,149.149
C06821=1125.859,-31.858,-48.749,179.570,5.759,149.150
C06822=1125.854,-31.609,-48.760,179.571,5.764,149.151
C06823=1125.848,-31.359,-48.772,179.570,5.768,149.152
C06824=1125.843,-31.109,-48.785,179.570,5.772,149.153
C06825=1125.839,-30.860,-48.796,179.570,5.776,149.154
C06826=1125.833,-30.610,-48.808,179.570,5.781,149.155
C06827=1125.828,-30.360,-48.820,179.570,5.785,149.156
C06828=1125.823,-30.110,-48.831,179.569,5.789,149.157
C06829=1125.818,-29.861,-48.844,179.569,5.793,149.158
C06830=1125.812,-29.612,-48.855,179.569,5.797,149.159
C06831=1125.806,-29.362,-48.867,179.569,5.801,149.160
C06832=1125.802,-29.112,-48.878,179.568,5.806,149.161
C06833=1125.796,-28.862,-48.890,179.568,5.810,149.162
C06834=1125.791,-28.613,-48.903,179.567,5.813,149.163
C06835=1125.786,-28.363,-48.915,179.566,5.818,149.164
C06836=1125.781,-28.113,-48.926,179.566,5.822,149.165
C06837=1125.776,-27.863,-48.938,179.565,5.826,149.166
C06838=1125.771,-27.614,-48.950,179.564,5.829,149.167
C06839=1125.765,-27.364,-48.962,179.563,5.834,149.169
C06840=1125.760,-27.114,-48.974,179.562,5.837,149.170
C06841=1125.755,-26.864,-48.985,179.561,5.842,149.171
C06842=1125.750,-26.615,-48.998,179.560,5.845,149.172
C06843=1125.744,-26.365,-49.010,179.560,5.849,149.173
C06844=1125.740,-26.116,-49.021,179.558,5.853,149.174
C06845=1125.735,-25.866,-49.034,179.558,5.858,149.175
C06846=1125.729,-25.616,-49.046,179.559,5.863,149.176
C06847=1125.723,-25.367,-49.057,179.560,5.868,149.177
C06848=1125.718,-25.117,-49.069,179.561,5.873,149.178
C06849=1125.713,-24.868,-49.081,179.561,5.878,149.179
C06850=1125.708,-24.618,-49.093,179.562,5.883,149.180
C06851=1125.703,-24.368,-49.105,179.563,5.888,149.180
C06852=1125.697,-24.119,-49.117,179.563,5.893,149.181
C06853=1125.692,-23.869,-49.129,179.565,5.898,149.182
C06854=1125.687,-23.620,-49.142,179.565,5.902,149.183
C06855=1125.681,-23.370,-49.154,179.566,5.907,149.184
C06856=1125.677,-23.120,-49.165,179.566,5.912,149.185
C06857=1125.672,-22.871,-49.178,179.567,5.917,149.186
C06858=1125.666,-22.621,-49.190,179.568,5.922,149.186
C06859=1125.661,-22.372,-49.202,179.569,5.927,149.187
C06860=1125.656,-22.122,-49.214,179.570,5.932,149.188
C06861=1125.650,-21.872,-49.226,179.571,5.937,149.189
C06862=1125.645,-21.622,-49.239,179.571,5.941,149.190
C06863=1125.640,-21.372,-49.250,179.572,5.946,149.190
C06864=1125.634,-21.123,-49.263,179.573,5.951,149.191
C06865=1125.630,-20.872,-49.275,179.574,5.956,149.192
C06866=1125.625,-20.658,-49.285,179.574,5.960,149.193
C06867=1125.620,-20.442,-49.296,179.575,5.964,149.194
C06868=1125.617,-20.227,-49.306,179.576,5.968,149.194
C06869=1125.612,-20.012,-49.318,179.576,5.972,149.195
C06870=1125.607,-19.796,-49.329,179.577,5.977,149.196
C06871=1125.603,-19.582,-49.339,179.578,5.981,149.196
C06872=1125.598,-19.366,-49.350,179.578,5.985,149.197
C06873=1125.594,-19.151,-49.360,179.578,5.989,149.198
C06874=1125.589,-18.901,-49.371,179.579,5.994,149.199
C06875=1125.584,-18.651,-49.384,179.580,5.998,149.200
C06876=1125.579,-18.401,-49.397,179.581,6.004,149.200
C06877=1125.574,-18.152,-49.409,179.582,6.008,149.201
C06878=1125.568,-17.902,-49.422,179.583,6.013,149.202
C06879=1125.562,-17.652,-49.434,179.583,6.018,149.203
C06880=1125.557,-17.403,-49.447,179.583,6.022,149.204
C06881=1125.552,-17.153,-49.459,179.584,6.027,149.204
C06882=1125.547,-16.903,-49.471,179.585,6.032,149.205
C06883=1125.542,-16.654,-49.484,179.586,6.037,149.206
C06884=1125.537,-16.404,-49.497,179.587,6.041,149.207
C06885=1125.532,-16.154,-49.509,179.588,6.046,149.208
C06886=1125.526,-15.905,-49.521,179.588,6.051,149.209
C06887=1125.521,-15.656,-49.534,179.589,6.055,149.209
C06888=1125.516,-15.406,-49.546,179.589,6.060,149.210
C06889=1125.511,-15.156,-49.558,179.590,6.065,149.211
C06890=1125.506,-14.906,-49.571,179.591,6.069,149.212
C06891=1125.501,-14.657,-49.584,179.592,6.075,149.213
C06892=1125.496,-14.407,-49.596,179.593,6.079,149.214
C06893=1125.490,-14.157,-49.609,179.594,6.084,149.214
C06894=1125.485,-13.908,-49.621,179.594,6.088,149.215
C06895=1125.480,-13.659,-49.634,179.595,6.093,149.216
C06896=1125.475,-13.408,-49.646,179.596,6.097,149.217
C06897=1125.470,-13.159,-49.659,179.596,6.102,149.218
C06898=1125.464,-12.909,-49.672,179.597,6.107,149.218
C06899=1125.459,-12.660,-49.684,179.598,6.111,149.219
C06900=1125.454,-12.410,-49.698,179.598,6.116,149.220
C06901=1125.449,-12.160,-49.710,179.599,6.121,149.221
C06902=1125.444,-11.911,-49.722,179.600,6.125,149.222
C06903=1125.438,-11.661,-49.735,179.600,6.130,149.222
C06904=1125.433,-11.412,-49.747,179.601,6.135,149.223
C06905=1125.428,-11.162,-49.761,179.601,6.139,149.224
C06906=1125.423,-10.912,-49.774,179.602,6.144,149.225
C06907=1125.418,-10.663,-49.786,179.603,6.148,149.226
C06908=1125.413,-10.414,-49.799,179.603,6.153,149.226
C06909=1125.408,-10.164,-49.812,179.604,6.157,149.227
C06910=1125.402,-9.914,-49.825,179.605,6.162,149.228
C06911=1125.397,-9.665,-49.838,179.605,6.166,149.229
C06912=1125.393,-9.415,-49.850,179.606,6.171,149.230
C06913=1125.388,-9.165,-49.863,179.607,6.176,149.231
C06914=1125.382,-8.916,-49.876,179.607,6.180,149.231
C06915=1125.376,-8.666,-49.888,179.608,6.185,149.232
C06916=1125.372,-8.416,-49.901,179.609,6.190,149.233
C06917=1125.367,-8.166,-49.914,179.610,6.194,149.234
C06918=1125.361,-7.917,-49.928,179.610,6.199,149.235
C06919=1125.357,-7.667,-49.941,179.611,6.204,149.235
C06920=1125.351,-7.418,-49.953,179.612,6.208,149.236
C06921=1125.346,-7.168,-49.966,179.612,6.213,149.237
C06922=1125.341,-6.953,-49.977,179.612,6.216,149.238
C06923=1125.337,-6.737,-49.989,179.613,6.221,149.238
C06924=1125.333,-6.522,-49.999,179.614,6.224,149.239
C06925=1125.328,-6.307,-50.011,179.614,6.229,149.240
C06926=1125.324,-6.091,-50.022,179.615,6.232,149.241
C06927=1125.319,-5.877,-50.033,179.615,6.236,149.241
C06928=1125.315,-5.661,-50.044,179.616,6.240,149.242
C06929=1125.310,-5.446,-50.056,179.616,6.244,149.243
C06930=1125.305,-5.196,-50.068,179.617,6.248,149.243
C06931=1125.299,-4.947,-50.081,179.618,6.253,149.244
C06932=1125.295,-4.697,-50.094,179.619,6.258,149.245
C06933=1125.289,-4.448,-50.108,179.619,6.262,149.246
C06934=1125.284,-4.198,-50.121,179.620,6.267,149.247
C06935=1125.280,-3.948,-50.134,179.620,6.271,149.247
C06936=1125.274,-3.699,-50.147,179.620,6.275,149.248
C06937=1125.269,-3.449,-50.160,179.621,6.280,149.249
C06938=1125.264,-3.199,-50.173,179.621,6.285,149.250
C06939=1125.259,-2.950,-50.187,179.622,6.289,149.251
C06940=1125.253,-2.700,-50.200,179.623,6.294,149.252
C06941=1125.248,-2.451,-50.213,179.624,6.298,149.252
C06942=1125.243,-2.201,-50.225,179.625,6.303,149.253
C06943=1125.238,-1.952,-50.240,179.625,6.308,149.254
C06944=1125.233,-1.702,-50.252,179.625,6.311,149.255
C06945=1125.228,-1.452,-50.266,179.626,6.316,149.256
C06946=1125.223,-1.203,-50.278,179.627,6.321,149.256
C06947=1125.218,-0.953,-50.293,179.627,6.325,149.257
C06948=1125.213,-0.704,-50.305,179.628,6.330,149.258
C06949=1125.207,-0.454,-50.318,179.628,6.335,149.259
C06950=1125.202,-0.204,-50.331,179.629,6.339,149.260
C06951=1125.197,0.045,-50.345,179.629,6.343,149.261
C06952=1125.192,0.295,-50.358,179.630,6.348,149.262
C06953=1125.186,0.545,-50.371,179.630,6.352,149.262
C06954=1125.182,0.794,-50.385,179.631,6.357,149.263
C06955=1125.176,1.044,-50.398,179.632,6.361,149.264
C06956=1125.172,1.294,-50.411,179.632,6.366,149.265
C06957=1125.166,1.543,-50.425,179.632,6.370,149.266
C06958=1125.162,1.793,-50.438,179.633,6.374,149.266
C06959=1125.156,2.042,-50.452,179.634,6.379,149.267
C06960=1125.150,2.291,-50.465,179.634,6.384,149.268
C06961=1125.146,2.541,-50.478,179.635,6.389,149.269
C06962=1125.140,2.790,-50.492,179.635,6.393,149.270
C06963=1125.136,3.040,-50.505,179.636,6.397,149.271
C06964=1125.130,3.289,-50.519,179.636,6.402,149.271
C06965=1125.125,3.540,-50.533,179.637,6.406,149.272
C06966=1125.120,3.789,-50.545,179.637,6.411,149.273
C06967=1125.115,4.039,-50.560,179.637,6.415,149.274
C06968=1125.110,4.288,-50.572,179.638,6.420,149.275
C06969=1125.105,4.538,-50.586,179.639,6.424,149.276
C06970=1125.099,4.788,-50.600,179.639,6.429,149.276
C06971=1125.095,5.037,-50.613,179.640,6.433,149.277
C06972=1125.089,5.287,-50.627,179.640,6.437,149.278
C06973=1125.084,5.536,-50.640,179.640,6.442,149.279
C06974=1125.079,5.786,-50.654,179.641,6.447,149.280
C06975=1125.074,6.035,-50.668,179.641,6.452,149.281
C06976=1125.069,6.285,-50.681,179.642,6.456,149.282
C06977=1125.064,6.534,-50.695,179.642,6.460,149.282
C06978=1125.059,6.750,-50.706,179.643,6.465,149.283
C06979=1125.055,6.965,-50.718,179.643,6.468,149.284
C06980=1125.050,7.180,-50.730,179.643,6.472,149.285
C06981=1125.046,7.396,-50.742,179.644,6.476,149.286
C06982=1125.042,7.611,-50.754,179.645,6.480,149.286
C06983=1125.037,7.825,-50.765,179.644,6.484,149.287
C06984=1125.032,8.041,-50.777,179.645,6.487,149.288
C06985=1125.028,8.256,-50.789,179.645,6.491,149.289
C06986=1125.024,8.506,-50.802,179.646,6.496,149.289
C06987=1125.018,8.755,-50.816,179.647,6.501,149.290
C06988=1125.013,9.005,-50.830,179.648,6.506,149.291
C06989=1125.008,9.254,-50.844,179.649,6.510,149.292
C06990=1125.003,9.504,-50.857,179.649,6.515,149.293
C06991=1124.998,9.754,-50.871,179.650,6.519,149.293
C06992=1124.993,10.003,-50.885,179.651,6.525,149.294
C06993=1124.987,10.253,-50.899,179.652,6.529,149.295
C06994=1124.982,10.502,-50.912,179.653,6.534,149.296
C06995=1124.977,10.752,-50.926,179.653,6.538,149.296
C06996=1124.973,11.001,-50.940,179.654,6.543,149.297
C06997=1124.967,11.251,-50.954,179.655,6.548,149.298
C06998=1124.962,11.501,-50.968,179.656,6.552,149.299
C06999=1124.957,11.750,-50.982,179.657,6.557,149.300
C07000=1124.952,11.999,-50.996,179.658,6.562,149.300
C07001=1124.947,12.249,-51.009,179.659,6.566,149.301
C07002=1124.942,12.499,-51.023,179.659,6.571,149.302
C07003=1124.936,12.748,-51.037,179.660,6.575,149.303
C07004=1124.931,12.998,-51.052,179.661,6.580,149.303
C07005=1124.926,13.247,-51.066,179.662,6.584,149.304
C07006=1124.920,13.497,-51.079,179.663,6.590,149.305
C07007=1124.916,13.746,-51.093,179.664,6.594,149.306
C07008=1124.911,13.996,-51.107,179.665,6.599,149.307
C07009=1124.906,14.245,-51.121,179.666,6.603,149.307
C07010=1124.901,14.495,-51.135,179.666,6.608,149.308
C07011=1124.896,14.745,-51.149,179.667,6.612,149.309
C07012=1124.891,14.994,-51.164,179.668,6.617,149.310
C07013=1124.885,15.243,-51.178,179.670,6.622,149.310
C07014=1124.880,15.494,-51.191,179.670,6.627,149.311
C07015=1124.875,15.743,-51.205,179.671,6.631,149.312
C07016=1124.870,15.993,-51.220,179.672,6.636,149.313
C07017=1124.865,16.242,-51.234,179.673,6.640,149.313
C07018=1124.860,16.492,-51.247,179.674,6.645,149.314
C07019=1124.855,16.741,-51.262,179.674,6.649,149.315
C07020=1124.850,16.991,-51.276,179.675,6.654,149.315
C07021=1124.845,17.240,-51.290,179.676,6.658,149.316
C07022=1124.840,17.490,-51.304,179.678,6.663,149.317
C07023=1124.835,17.739,-51.318,179.679,6.668,149.318
C07024=1124.830,17.989,-51.333,179.679,6.672,149.319
C07025=1124.824,18.238,-51.347,179.680,6.677,149.319
C07026=1124.819,18.488,-51.361,179.681,6.681,149.320
C07027=1124.815,18.738,-51.375,179.682,6.686,149.321
C07028=1124.810,18.987,-51.389,179.683,6.690,149.321
C07029=1124.805,19.237,-51.404,179.684,6.694,149.322
C07030=1124.798,19.486,-51.418,179.684,6.699,149.323
C07031=1124.793,19.736,-51.432,179.686,6.704,149.324
C07032=1124.789,19.985,-51.447,179.687,6.708,149.324
C07033=1124.784,20.235,-51.462,179.688,6.713,149.325
C07034=1124.780,20.450,-51.473,179.689,6.716,149.325
C07035=1124.775,20.665,-51.486,179.690,6.721,149.326
C07036=1124.771,20.880,-51.498,179.690,6.724,149.327
C07037=1124.766,21.095,-51.511,179.691,6.729,149.327
C07038=1124.762,21.310,-51.523,179.692,6.732,149.328
C07039=1124.757,21.525,-51.536,179.693,6.736,149.329
C07040=1124.754,21.740,-51.548,179.694,6.740,149.329
C07041=1124.749,21.956,-51.560,179.695,6.744,149.330
C07042=1124.744,22.205,-51.575,179.696,6.748,149.330
C07043=1124.739,22.454,-51.590,179.697,6.753,149.331
C07044=1124.734,22.704,-51.604,179.697,6.757,149.332
C07045=1124.729,22.953,-51.618,179.698,6.762,149.333
C07046=1124.723,23.203,-51.633,179.699,6.766,149.333
C07047=1124.718,23.453,-51.647,179.700,6.770,149.334
C07048=1124.713,23.702,-51.662,179.701,6.775,149.335
C07049=1124.708,23.952,-51.676,179.702,6.779,149.335
C07050=1124.703,24.201,-51.691,179.703,6.784,149.336
C07051=1124.698,24.451,-51.705,179.704,6.788,149.337
C07052=1124.693,24.701,-51.720,179.705,6.792,149.337
C07053=1124.688,24.950,-51.735,179.706,6.797,149.338
C07054=1124.683,25.200,-51.749,179.707,6.801,149.339
C07055=1124.678,25.448,-51.764,179.708,6.805,149.339
C07056=1124.673,25.698,-51.778,179.710,6.811,149.340
C07057=1124.667,25.948,-51.793,179.711,6.815,149.341
C07058=1124.663,26.197,-51.808,179.712,6.819,149.342
C07059=1124.658,26.447,-51.822,179.713,6.824,149.342
C07060=1124.653,26.696,-51.837,179.714,6.828,149.343
C07061=1124.647,26.946,-51.852,179.715,6.832,149.343
C07062=1124.642,27.196,-51.866,179.716,6.837,149.344
C07063=1124.638,27.445,-51.881,179.717,6.841,149.345
C07064=1124.632,27.695,-51.896,179.718,6.845,149.345
C07065=1124.627,27.944,-51.911,179.719,6.850,149.346
C07066=1124.622,28.194,-51.925,179.720,6.854,149.347
C07067=1124.617,28.443,-51.940,179.721,6.858,149.347
C07068=1124.612,28.693,-51.955,179.722,6.862,149.348
C07069=1124.607,28.942,-51.969,179.723,6.867,149.349
C07070=1124.602,29.192,-51.984,179.724,6.871,149.349
C07071=1124.597,29.442,-51.999,179.725,6.876,149.350
C07072=1124.592,29.691,-52.014,179.726,6.880,149.351
C07073=1124.587,29.940,-52.029,179.727,6.884,149.351
C07074=1124.582,30.190,-52.044,179.728,6.889,149.352
C07075=1124.577,30.439,-52.058,179.729,6.893,149.353
C07076=1124.572,30.689,-52.073,179.730,6.897,149.353
C07077=1124.567,30.938,-52.089,179.732,6.901,149.354
C07078=1124.562,31.188,-52.103,179.733,6.906,149.355
C07079=1124.556,31.437,-52.119,179.734,6.910,149.355
C07080=1124.551,31.687,-52.133,179.735,6.914,149.356
C07081=1124.547,31.936,-52.148,179.736,6.919,149.356
C07082=1124.541,32.185,-52.164,179.737,6.923,149.357
C07083=1124.536,32.435,-52.178,179.738,6.927,149.358
C07084=1124.531,32.684,-52.194,179.739,6.932,149.358
C07085=1124.526,32.934,-52.208,179.740,6.936,149.359
C07086=1124.521,33.184,-52.224,179.741,6.940,149.360
C07087=1124.517,33.433,-52.239,179.742,6.944,149.360
C07088=1124.512,33.683,-52.253,179.743,6.949,149.361
C07089=1124.506,33.932,-52.269,179.744,6.953,149.362
C07090=1124.502,34.147,-52.282,179.746,6.957,149.362
C07091=1124.497,34.362,-52.295,179.746,6.961,149.363
C07092=1124.493,34.577,-52.307,179.748,6.964,149.363
C07093=1124.489,34.793,-52.320,179.748,6.968,149.364
C07094=1124.485,35.008,-52.333,179.750,6.972,149.364
C07095=1124.480,35.222,-52.347,179.750,6.975,149.365
C07096=1124.476,35.437,-52.360,179.751,6.979,149.365
C07097=1124.471,35.652,-52.373,179.752,6.983,149.366
C07098=1124.467,35.902,-52.388,179.754,6.987,149.366
C07099=1124.461,36.152,-52.403,179.755,6.991,149.367
C07100=1124.457,36.401,-52.418,179.756,6.995,149.368
C07101=1124.451,36.650,-52.434,179.757,7.000,149.368
C07102=1124.446,36.900,-52.450,179.758,7.004,149.369
C07103=1124.441,37.149,-52.464,179.759,7.008,149.370
C07104=1124.436,37.399,-52.479,179.761,7.012,149.370
C07105=1124.432,37.648,-52.495,179.762,7.017,149.371
C07106=1124.426,37.898,-52.510,179.763,7.021,149.371
C07107=1124.422,38.147,-52.525,179.764,7.025,149.372
C07108=1124.416,38.396,-52.541,179.765,7.029,149.373
C07109=1124.411,38.646,-52.556,179.767,7.033,149.373
C07110=1124.406,38.895,-52.571,179.768,7.038,149.374
C07111=1124.401,39.146,-52.587,179.769,7.042,149.374
C07112=1124.396,39.395,-52.602,179.770,7.046,149.375
C07113=1124.391,39.644,-52.617,179.771,7.050,149.375
C07114=1124.386,39.893,-52.633,179.772,7.055,149.376
C07115=1124.381,40.143,-52.648,179.773,7.059,149.377
C07116=1124.376,40.393,-52.664,179.775,7.063,149.377
C07117=1124.371,40.642,-52.679,179.776,7.067,149.378
C07118=1124.366,40.891,-52.694,179.777,7.071,149.378
C07119=1124.361,41.141,-52.710,179.778,7.076,149.379
C07120=1124.356,41.391,-52.726,179.779,7.080,149.380
C07121=1124.351,41.640,-52.741,179.780,7.083,149.380
C07122=1124.346,41.889,-52.757,179.781,7.087,149.381
C07123=1124.341,42.139,-52.772,179.782,7.092,149.381
C07124=1124.335,42.388,-52.788,179.784,7.096,149.382
C07125=1124.331,42.638,-52.803,179.785,7.100,149.383
C07126=1124.326,42.887,-52.819,179.786,7.104,149.383
C07127=1124.320,43.137,-52.834,179.787,7.109,149.384
C07128=1124.316,43.387,-52.850,179.789,7.113,149.384
C07129=1124.311,43.635,-52.866,179.790,7.117,149.385
C07130=1124.306,43.884,-52.882,179.791,7.121,149.386
C07131=1124.300,44.134,-52.897,179.792,7.125,149.386
C07132=1124.296,44.384,-52.913,179.793,7.129,149.387
C07133=1124.291,44.633,-52.928,179.795,7.134,149.387
C07134=1124.286,44.882,-52.944,179.796,7.138,149.388
C07135=1124.281,45.133,-52.960,179.797,7.142,149.388
C07136=1124.275,45.382,-52.975,179.798,7.146,149.389
C07137=1124.270,45.631,-52.991,179.800,7.150,149.389
C07138=1124.266,45.881,-53.007,179.801,7.154,149.390
C07139=1124.261,46.130,-53.022,179.802,7.158,149.391
C07140=1124.256,46.379,-53.038,179.804,7.163,149.391
C07141=1124.251,46.629,-53.054,179.805,7.167,149.392
C07142=1124.246,46.878,-53.070,179.806,7.171,149.392
C07143=1124.241,47.127,-53.085,179.807,7.175,149.393
C07144=1124.236,47.377,-53.101,179.809,7.179,149.393
C07145=1124.231,47.627,-53.117,179.810,7.183,149.394
C07146=1124.227,47.841,-53.131,179.811,7.187,149.394
C07147=1124.222,48.057,-53.145,179.811,7.190,149.395
C07148=1124.218,48.271,-53.158,179.813,7.194,149.395
C07149=1124.214,48.487,-53.172,179.814,7.197,149.396
C07150=1124.210,48.701,-53.186,179.815,7.201,149.396
C07151=1124.205,48.916,-53.199,179.816,7.204,149.397
C07152=1124.201,49.131,-53.213,179.817,7.208,149.397
C07153=1124.196,49.346,-53.227,179.818,7.212,149.398
C07154=1124.192,49.595,-53.243,179.820,7.215,149.398
C07155=1124.187,49.845,-53.258,179.821,7.220,149.399
C07156=1124.182,50.094,-53.275,179.822,7.224,149.400
C07157=1124.177,50.344,-53.291,179.824,7.228,149.400
C07158=1124.172,50.593,-53.306,179.825,7.232,149.401
C07159=1124.167,50.842,-53.323,179.826,7.236,149.401
C07160=1124.162,51.092,-53.338,179.827,7.240,149.402
C07161=1124.157,51.341,-53.355,179.828,7.244,149.402
C07162=1124.152,51.591,-53.371,179.829,7.248,149.403
C07163=1124.147,51.841,-53.387,179.831,7.252,149.403
C07164=1124.142,52.090,-53.403,179.832,7.256,149.404
C07165=1124.137,52.339,-53.418,179.833,7.260,149.404
C07166=1124.132,52.589,-53.435,179.835,7.264,149.405
C07167=1124.127,52.838,-53.451,179.836,7.268,149.405
C07168=1124.122,53.087,-53.467,179.837,7.273,149.406
C07169=1124.117,53.337,-53.483,179.839,7.276,149.406
C07170=1124.112,53.586,-53.500,179.840,7.281,149.407
C07171=1124.107,53.836,-53.515,179.841,7.285,149.407
C07172=1124.102,54.085,-53.532,179.843,7.289,149.408
C07173=1124.096,54.335,-53.548,179.844,7.293,149.409
C07174=1124.092,54.584,-53.565,179.845,7.297,149.409
C07175=1124.087,54.833,-53.581,179.847,7.301,149.410
C07176=1124.082,55.083,-53.597,179.848,7.305,149.410
C07177=1124.077,55.332,-53.613,179.849,7.309,149.411
C07178=1124.072,55.582,-53.629,179.850,7.314,149.411
C07179=1124.067,55.831,-53.646,179.852,7.318,149.412
C07180=1124.063,56.080,-53.662,179.852,7.321,149.412
C07181=1124.057,56.330,-53.678,179.854,7.325,149.413
C07182=1124.053,56.579,-53.695,179.856,7.329,149.413
C07183=1124.047,56.828,-53.711,179.857,7.333,149.414
C07184=1124.042,57.079,-53.727,179.858,7.337,149.414
C07185=1124.037,57.327,-53.744,179.859,7.341,149.415
C07186=1124.033,57.577,-53.760,179.861,7.345,149.415
C07187=1124.028,57.827,-53.776,179.862,7.350,149.416
C07188=1124.023,58.076,-53.793,179.864,7.353,149.417
C07189=1124.017,58.325,-53.810,179.865,7.357,149.417
C07190=1124.012,58.575,-53.825,179.866,7.362,149.418
C07191=1124.008,58.824,-53.842,179.868,7.366,149.418
C07192=1124.002,59.073,-53.858,179.869,7.370,149.419
C07193=1123.998,59.323,-53.875,179.870,7.374,149.419
C07194=1123.993,59.572,-53.892,179.872,7.378,149.420
C07195=1123.987,59.822,-53.908,179.873,7.382,149.420
C07196=1123.983,60.071,-53.925,179.875,7.386,149.421
C07197=1123.978,60.320,-53.941,179.875,7.389,149.421
C07198=1123.973,60.570,-53.958,179.877,7.393,149.422
C07199=1123.968,60.819,-53.975,179.878,7.397,149.422
C07200=1123.963,61.069,-53.990,179.879,7.402,149.423
C07201=1123.958,61.318,-54.007,179.881,7.405,149.423
C07202=1123.953,61.533,-54.021,179.883,7.409,149.424
C07203=1123.950,61.747,-54.036,179.883,7.412,149.424
C07204=1123.945,61.963,-54.051,179.884,7.416,149.424
C07205=1123.941,62.177,-54.065,179.886,7.420,149.425
C07206=1123.937,62.392,-54.079,179.887,7.423,149.425
C07207=1123.932,62.607,-54.093,179.888,7.427,149.426
C07208=1123.928,62.822,-54.108,179.889,7.430,149.426
C07209=1123.925,63.036,-54.122,179.890,7.433,149.427
C07210=1123.918,63.286,-54.139,179.891,7.437,149.427
C07211=1123.914,63.536,-54.155,179.893,7.441,149.428
C07212=1123.909,63.785,-54.172,179.894,7.445,149.428
C07213=1123.904,64.034,-54.189,179.896,7.449,149.429
C07214=1123.899,64.284,-54.205,179.897,7.453,149.429
C07215=1123.894,64.533,-54.223,179.898,7.457,149.430
C07216=1123.889,64.783,-54.239,179.900,7.461,149.430
C07217=1123.884,65.032,-54.256,179.902,7.465,149.431
C07218=1123.879,65.282,-54.273,179.903,7.469,149.431
C07219=1123.875,65.531,-54.290,179.904,7.473,149.432
C07220=1123.870,65.780,-54.306,179.906,7.477,149.432
C07221=1123.865,66.029,-54.324,179.907,7.482,149.433
C07222=1123.860,66.278,-54.341,179.908,7.486,149.433
C07223=1123.855,66.528,-54.358,179.910,7.489,149.434
C07224=1123.850,66.777,-54.374,179.911,7.494,149.434
C07225=1123.845,67.027,-54.391,179.913,7.498,149.435
C07226=1123.840,67.276,-54.408,179.914,7.501,149.435
C07227=1123.836,67.526,-54.425,179.915,7.505,149.436
C07228=1123.830,67.775,-54.442,179.916,7.509,149.436
C07229=1123.825,68.024,-54.458,179.918,7.513,149.437
C07230=1123.821,68.274,-54.476,179.919,7.517,149.437
C07231=1123.816,68.523,-54.493,179.921,7.521,149.438
C07232=1123.810,68.772,-54.510,179.922,7.525,149.438
C07233=1123.806,69.022,-54.527,179.924,7.529,149.439
C07234=1123.801,69.271,-54.544,179.925,7.533,149.439
C07235=1123.796,69.520,-54.561,179.926,7.537,149.440
C07236=1123.791,69.770,-54.578,179.928,7.541,149.440
C07237=1123.786,70.019,-54.595,179.930,7.545,149.441
C07238=1123.781,70.269,-54.612,179.931,7.549,149.441
C07239=1123.776,70.518,-54.629,179.932,7.553,149.442
C07240=1123.771,70.767,-54.647,179.934,7.557,149.442
C07241=1123.766,71.017,-54.664,179.935,7.561,149.443
C07242=1123.761,71.266,-54.680,179.937,7.565,149.443
C07243=1123.756,71.515,-54.698,179.938,7.569,149.444
C07244=1123.752,71.765,-54.715,179.940,7.573,149.444
C07245=1123.747,72.014,-54.732,179.941,7.577,149.445
C07246=1123.742,72.264,-54.750,179.942,7.581,149.445
C07247=1123.737,72.513,-54.767,179.943,7.584,149.445
C07248=1123.732,72.763,-54.784,179.945,7.588,149.446
C07249=1123.727,73.011,-54.801,179.946,7.592,149.447
C07250=1123.722,73.261,-54.818,179.948,7.596,149.447
C07251=1123.717,73.511,-54.836,179.949,7.600,149.447
C07252=1123.713,73.759,-54.853,179.951,7.604,149.448
C07253=1123.707,74.009,-54.870,179.952,7.608,149.448
C07254=1123.702,74.258,-54.888,179.953,7.612,149.449
C07255=1123.698,74.508,-54.905,179.955,7.616,149.449
C07256=1123.693,74.757,-54.923,179.957,7.620,149.450
C07257=1123.687,75.006,-54.940,179.958,7.624,149.450
C07258=1123.683,75.221,-54.955,179.959,7.628,149.451
C07259=1123.679,75.436,-54.969,179.960,7.631,149.451
C07260=1123.675,75.651,-54.985,179.962,7.634,149.451
C07261=1123.671,75.865,-55.000,179.963,7.638,149.452
C07262=1123.666,76.080,-55.014,179.964,7.641,149.452
C07263=1123.662,76.295,-55.030,179.966,7.645,149.453
C07264=1123.658,76.509,-55.045,179.967,7.648,149.453
C07265=1123.654,76.724,-55.060,179.968,7.651,149.454
C07266=1123.649,76.974,-55.077,179.969,7.656,149.454
C07267=1123.644,77.223,-55.095,179.970,7.659,149.455
C07268=1123.639,77.473,-55.112,179.971,7.663,149.455
C07269=1123.634,77.722,-55.130,179.972,7.666,149.456
C07270=1123.630,77.971,-55.147,179.973,7.670,149.456
C07271=1123.625,78.220,-55.165,179.974,7.674,149.457
C07272=1123.620,78.470,-55.183,179.974,7.677,149.457
C07273=1123.615,78.719,-55.200,179.976,7.681,149.458
C07274=1123.611,78.968,-55.218,179.977,7.684,149.459
C07275=1123.605,79.217,-55.235,179.978,7.689,149.459
C07276=1123.600,79.467,-55.253,179.979,7.692,149.460
C07277=1123.595,79.716,-55.271,179.980,7.696,149.460
C07278=1123.590,79.966,-55.288,179.981,7.700,149.461
C07279=1123.585,80.215,-55.306,179.982,7.703,149.461
C07280=1123.581,80.464,-55.323,179.983,7.707,149.462
C07281=1123.575,80.713,-55.340,179.984,7.711,149.462
C07282=1123.570,80.963,-55.358,179.986,7.715,149.463
C07283=1123.566,81.212,-55.376,179.986,7.718,149.463
C07284=1123.560,81.462,-55.394,179.988,7.722,149.464
C07285=1123.556,81.711,-55.412,179.989,7.726,149.465
C07286=1123.551,81.961,-55.430,179.990,7.730,149.465
C07287=1123.547,82.209,-55.447,179.991,7.734,149.466
C07288=1123.542,82.459,-55.465,179.992,7.737,149.466
C07289=1123.537,82.708,-55.483,179.993,7.741,149.467
C07290=1123.532,82.958,-55.501,179.995,7.745,149.467
C07291=1123.527,83.207,-55.519,179.996,7.748,149.468
C07292=1123.522,83.457,-55.536,179.997,7.753,149.468
C07293=1123.517,83.706,-55.554,179.998,7.756,149.469
C07294=1123.512,83.955,-55.572,179.999,7.760,149.469
C07295=1123.507,84.204,-55.590,-180.000,7.764,149.470
C07296=1123.502,84.453,-55.608,-179.999,7.768,149.470
C07297=1123.497,84.702,-55.626,-179.998,7.771,149.471
C07298=1123.492,84.952,-55.643,-179.996,7.775,149.471
C07299=1123.487,85.201,-55.661,-179.995,7.779,149.472
C07300=1123.483,85.450,-55.678,-179.993,7.783,149.472
C07301=1123.478,85.699,-55.696,-179.992,7.786,149.473
C07302=1123.474,85.949,-55.715,-179.991,7.791,149.473
C07303=1123.469,86.198,-55.733,-179.990,7.795,149.474
C07304=1123.464,86.448,-55.751,-179.988,7.798,149.474
C07305=1123.459,86.697,-55.769,-179.987,7.803,149.475
C07306=1123.454,86.946,-55.787,-179.986,7.806,149.475
C07307=1123.449,87.196,-55.804,-179.984,7.810,149.476
C07308=1123.443,87.445,-55.822,-179.983,7.814,149.476
C07309=1123.438,87.694,-55.840,-179.982,7.818,149.477
C07310=1123.434,87.944,-55.859,-179.980,7.822,149.477
C07311=1123.429,88.194,-55.877,-179.979,7.825,149.478
C07312=1123.424,88.443,-55.895,-179.977,7.829,149.478
C07313=1123.419,88.692,-55.913,-179.976,7.833,149.479
C07314=1123.415,88.906,-55.929,-179.975,7.836,149.479
C07315=1123.411,89.121,-55.944,-179.973,7.840,149.479
C07316=1123.407,89.335,-55.960,-179.972,7.843,149.480
C07317=1123.403,89.550,-55.975,-179.971,7.846,149.480
C07318=1123.399,89.765,-55.990,-179.970,7.850,149.481
C07319=1123.394,89.980,-56.006,-179.969,7.853,149.481
C07320=1123.390,90.194,-56.022,-179.968,7.856,149.481
